DATA_BLOCK "Asse_B"	// DB 35
VERSION : 0.1
  STRUCT
   A_FD_OR : BYTE ;	//Feedrate override
   A_DriveEnable : BOOL ;	//Drive test movement enable
   A_AckFixedStop : BOOL ;	//Acknowledge fixed stop reached
   A_SensorFixedStop : BOOL ;	//Sensor fixed stop
   A_ASpDisable : BOOL ;	//Axis/spindle disable
   A_Follow_upMode : BOOL ;	//Follow-up mode
   A_PosMeas1 : BOOL ;	//Position measuring system 1
   A_PosMeas2 : BOOL ;	//Position measuring system 2
   A_ORactive : BOOL ;	//Override active
   A_SWCam : BOOL ;	//SW cam activation
   A_ContrEnable : BOOL ;	//Controller enable
   A_DelDTGSpReset : BOOL ;	//Delete distance to go/Spindle-Reset
   A_Clamp : BOOL ;	//Clamping in progress
   A_RefVal1 : BOOL ;	//Reference point value 1
   A_RefVal2 : BOOL ;	//Reference point value 2
   A_RefVal3 : BOOL ;	//Reference point value 3
   A_RefVal4 : BOOL ;	//Reference point value 4
   A_ExtZO : BOOL ;	//Import external ZO
   A_EnabTravFixedStop : BOOL ;	//Enable travel to fixed stop
   A_FixedFD1 : BOOL ;	//Activate fixed feed 1
   A_FixedFD2 : BOOL ;	//Activate fixed feed 2
   A_FixedFD3 : BOOL ;	//Activate fixed feed 3
   A_FixedFD4 : BOOL ;	//Activate fixed feed 4
   A_VelocSpeedLimit : BOOL ;	//Velocity/spindle speed limitation
   A_PrgtestAxRel : BOOL ;	// Program test axis/spindle release
   A_HW1 : BOOL ;	//Activate handwheel 1
   A_HW2 : BOOL ;	//Activate handwheel 2
   A_HW3 : BOOL ;	//Activate handwheel 3
   A_FDSpStop : BOOL ;	//Feed stop/spindle stop
   A_Disable : BOOL ;	//Traversing key disable
   A_RapidTrOR : BOOL ;	//Rapid traverse override
   A_Minus : BOOL ;	//Traversing key minus
   A_Plus : BOOL ;	//Traversing key plus
   A_INC1 : BOOL ;	//INC1
   A_INC10 : BOOL ;	//INC10
   A_INC100 : BOOL ;	//INC100
   A_INC1000 : BOOL ;	//INC1000
   A_INC10000 : BOOL ;	//INC10000
   A_INCVar : BOOL ;	//INC variable
   A_OEMAxis : BYTE ;	//OEM axis signals
   f7 : BYTE ;
   A_NCASpChanA : BOOL ;	//Assign NC axis/spindle channel A
   A_NCASpChanB : BOOL ;	//Assign NC axis/spindle channel B
   A_NCASpChanC : BOOL ;	//Assign NC axis/spindle channel C
   A_NCASpChanD : BOOL ;	//Assign NC axis/spindle channel D
   A_NCASpStrobe : BOOL ;	//Activation of assignment with pos. edge
   f8_5 : BOOL ;
   f8_6 : BOOL ;
   A_PLCASp : BOOL ;	//Request PLC axis/spindle
   A_Para_A : BOOL ;	//Parameter block servo A
   A_Para_B : BOOL ;	//Parameter block servo B
   A_Para_C : BOOL ;	//Parameter block servo C
   A_LockParSetDef : BOOL ;	//Lock parameter set definition from NC
   f9_4 : BOOL ;
   f9_5 : BOOL ;
   f9_6 : BOOL ;
   f9_7 : BOOL ;
   A_REPOSDelay : BOOL ;	//REPOS DELAY
   f10_1 : BOOL ;
   f10_2 : BOOL ;
   f10_3 : BOOL ;
   f10_4 : BOOL ;
   f10_5 : BOOL ;
   f10_6 : BOOL ;
   f10_7 : BOOL ;
   A_StartBrakeTest : BOOL ;	// Start brake test
   f11_1 : BOOL ;
   f11_2 : BOOL ;
   f11_3 : BOOL ;
   f11_4 : BOOL ;
   f11_5 : BOOL ;
   f11_6 : BOOL ;
   f11_7 : BOOL ;
   A_HWLimitMinus : BOOL ;	//Hardware limit switch minus
   A_HWLimitPlus : BOOL ;	//Hardware limit switch plus
   A_SWLimit2Minus : BOOL ;	//2nd software limit switch minus
   A_SWLimit2Plus : BOOL ;	//2nd software limit switch plus
   A_ModuloLimitEn : BOOL ;	// Modulo limit enabled
   f12_5 : BOOL ;
   f12_6 : BOOL ;
   A_DelayRef : BOOL ;	//Delay reference point approach
   f13 : BYTE ;
   f14 : INT ;
   A_ActGearA : BOOL ;	//Actual gear stage A
   A_ActGearB : BOOL ;	//Actual gear stage B
   A_ActGearC : BOOL ;	//Actual gear stage C
   A_GearChangeOv : BOOL ;	//Gear has changed over
   A_Sp1Syn : BOOL ;	//Re-synchronize spindle 1
   A_Sp2Syn : BOOL ;	//Re-synchronize spindle 2
   A_NoMonitorGear : BOOL ;	//No monitoring when changing gear
   A_DeleteS : BOOL ;	//Delete S value
   A_FD_ORSp : BOOL ;	//Feedrate override for spindle valid
   f17_1 : BOOL ;
   f17_2 : BOOL ;
   f17_3 : BOOL ;
   A_Sp1SynP : BOOL ;	//Re-synchronize spindle 1 f. positioning
   A_Sp2SynP : BOOL ;	//Re-synchronize spindle 2 f. positioning
   A_M3M4Inv : BOOL ;	//Invert M3/M4
   f17_7 : BOOL ;
   f18_0 : BOOL ;
   f18_1 : BOOL ;
   f18_2 : BOOL ;
   f18_3 : BOOL ;
   A_OscilPLC : BOOL ;	//Oscillation via PLC
   A_OscilSpeed : BOOL ;	//enable Oscillation
   A_SetRotDirectRight : BOOL ;	//Setpoint osci. direct. right
   A_SetRotDirectLeft : BOOL ;	//Setpoint osci. direct. left
   A_SpOR : BYTE ;	//Spindle override
   A_UFSwOv : BOOL ;	//Run-up switchover U/F operation
   A_RUEncQuStop : BOOL ;	//Run-up encoder quick stop
   A_Tlimit2 : BOOL ;	//Torque limit 2
   A_SpeedSetpSmooth : BOOL ;	//Speed setpoint smoothing
   f20_4 : BOOL ;
   A_HoldBrakeToOpen : BOOL ;	// holding brake open
   f20_6 : BOOL ;
   f20_7 : BOOL ;
   A_ParA : BOOL ;	//Parameter set selection A
   A_ParB : BOOL ;	//Parameter set selection B
   A_ParC : BOOL ;	//Parameter set selection C
   A_MotA : BOOL ;	//Motor selection A
   A_MotB : BOOL ;	//Motor selection B
   A_MotOK : BOOL ;	//Motor selected
   A_IntegratDisable : BOOL ;	//n controller integrator disable
   A_PulseEnable : BOOL ;	//Pulse enable
   A_SG_SBH : BOOL ;	//Deselection SG/SBH
   A_SBH : BOOL ;	//Deselection of safe standstill
   f22_2 : BOOL ;
   A_SGselect0 : BOOL ;	//Selection SG bit 0
   A_SGselect1 : BOOL ;	//Selection SG bit 1
   f22_5 : BOOL ;
   f22_6 : BOOL ;
   f22_7 : BOOL ;
   A_Transmiss0 : BOOL ;	//Selection Transmission bit 0
   A_Transmiss1 : BOOL ;	//Selection Transmission bit 1
   A_Transmiss2 : BOOL ;	//Selection Transmission bit 2
   f23_3 : BOOL ;
   A_SE : BOOL ;	//Selection SE
   A_BrakeToClose : BOOL ;	// Sinamics: Brake to close
   f23_6 : BOOL ;
   A_TestStop : BOOL ;	//Activate test stop
   A_RotationMonit : BOOL ;	// Stepper motor: Rotation monitoring
   A_ControlAx : BOOL ;	// Control Axis
   f24_2 : BOOL ;
   f24_3 : BOOL ;
   A_TorqComp : BOOL ;	// Torque compensation
   A_ChangSetpOutAss0 : BOOL ;	// Bit value for CTRLOUT_changed - Change setpoint output assignment
   A_ChangSetpOutAss1 : BOOL ;	// Bit value for CTRLOUT_changed - Change setpoint output assignment
   A_MS : BOOL ;	//Master / Slave On
   f25 : BYTE ;
   f26_0 : BOOL ;
   f26_1 : BOOL ;
   f26_2 : BOOL ;
   A_CompContr : BOOL ;	//Compensation controller On
   A_FollowAxOv : BOOL ;	//Enable following axis override
   f26_5 : BOOL ;
   f26_6 : BOOL ;
   f26_7 : BOOL ;
   A_DEPMCS : BOOL ;	// Resume: DEPMCS
   A_DEPBCS : BOOL ;	// Resume: DEPBCS
   A_Corr : BOOL ;	// Resume: Corr
   A_HIAxMove : BOOL ;	// Resume: HIAxMove
   A_StopDEPMCS : BOOL ;	// Stop: DEPMCS
   A_StopDEPBCS : BOOL ;	// Stop: DEPBCS
   A_StopCorr : BOOL ;	// Stop: Corr
   A_StopHIAxMove : BOOL ;	// Stop: HIAxMove
   A_OscillAxExtRev : BOOL ;	// OscillAxExtReversal
   A_AxReset : BOOL ;	// AXRESET
   A_AxResume : BOOL ;	// AXRESUME
   A_SetRP : BOOL ;	//Set reversal point
   A_ChangeRP : BOOL ;	//Change reversal point
   A_StopRP : BOOL ;	//Stop at next reversal point
   A_Stop : BOOL ;	//Stop
   A_PLCAxis : BOOL ;	//PLC checks axis
   f29_0 : BOOL ;
   f29_1 : BOOL ;
   f29_2 : BOOL ;
   f29_3 : BOOL ;
   A_StartGantSynRun : BOOL ;	//Start gantry synchronization run
   A_NoAutoSync : BOOL ;	//No auto sync
   f29_6 : BOOL ;
   f29_7 : BOOL ;
   A_StopSpindle : BOOL ;	//Stop spindle
   A_StartCW : BOOL ;	//Start spindle Clockwise
   A_StartCCW : BOOL ;	//Start spindle Counterclockwise
   A_AutoGearStep : BOOL ;	//Autom. gear step change
   A_PosSpindle : BOOL ;	//Position spindle
   f30_5 : BOOL ;
   f30_6 : BOOL ;
   f30_7 : BOOL ;
   f31_0 : BOOL ;
   f31_1 : BOOL ;
   f31_2 : BOOL ;
   f31_3 : BOOL ;
   A_Resynchronize : BOOL ;	// Resynchronize
   A_DisSync : BOOL ;	// Disable synchronization
   A_Tracksync : BOOL ;	// Track synchronism
   f31_7 : BOOL ;
   f32_0 : BOOL ;
   f32_1 : BOOL ;
   A_extStopA : BOOL ;	//Deselection external Stop A
   A_extStopC : BOOL ;	//Deselection external Stop C
   A_extStopD : BOOL ;	//Deselection external Stop D
   A_extStopE : BOOL ;	//Deselection external Stop E
   f32_6 : BOOL ;
   f32_7 : BOOL ;
   f33_0 : BOOL ;
   f33_1 : BOOL ;
   f33_2 : BOOL ;
   f33_3 : BOOL ;
   A_SGcorr_0 : BOOL ;	//Selection SG-correction Bit 0
   A_SGcorr_1 : BOOL ;	//Selection SG-correction Bit 1
   A_SGcorr_2 : BOOL ;	//Selection SG-correction Bit 2
   A_SGcorr_3 : BOOL ;	//Selection SG-correction Bit 3
   f34 : ARRAY  [34 .. 55 ] OF BYTE ;
   A_FeedDriveCAxEng : BOOL ;	// Seperate feed drive as C axis engaged
   A_SpSpeedDisp : BOOL ;	// Spindle speed display
   A_SpInsideClamp : BOOL ;	// Spindle inside clamping
   f56_3 : BOOL ;
   f56_4 : BOOL ;
   f56_5 : BOOL ;
   f56_6 : BOOL ;
   f56_7 : BOOL ;
   f57 : BYTE ;
   f58 : WORD ;	// FC18: internal
   E_SpNA : BOOL ;	//Spindle/no axis
   E_NCU_Link : BOOL ;	//NCU_link active axis
   E_EncodFreq1 : BOOL ;	//Encoder limit frequency 1 exceeded
   E_EncodFreq2 : BOOL ;	//Encoder limit frequency 2 exceeded
   E_RefSyn1 : BOOL ;	//Referenced/synchronized 1
   E_RefSyn2 : BOOL ;	//Referenced/synchronized 2
   E_ExactCoarse : BOOL ;	//Position reached with exact stop coarse
   E_ExactFine : BOOL ;	//Position reached with exact stop fine
   E_TravRequ : BOOL ;	//Travel request
   E_AxialAlarm : BOOL ;	// Axial alarm
   E_AxisReady : BOOL ;	//Axis ready
   E_Follow_upMode : BOOL ;	//Follow-up mode active
   E_Stat : BOOL ;	//Axis/spindle stationary (n<nmin)
   E_PositContr : BOOL ;	//Position controller active
   E_SpeedContr : BOOL ;	//Speed controller active
   E_CurrentContr : BOOL ;	//Current controller active
   E_SWCam : BOOL ;	//Software cams active
   E_HWOverlay : BOOL ;	//Handwheel overlay active
   E_RevFD : BOOL ;	//Revolutional feedrate active
   E_MeasAct : BOOL ;	//Measuring active
   E_ActTravFStop : BOOL ;	//Activate travel to fixed stop
   E_FixedStop : BOOL ;	//Fixed stop reached
   E_ForceFixedStop : BOOL ;	// Force fixed stop limited
   E_AxContainerRot : BOOL ;	// Axis container rotation active
   E_AxReset : BOOL ;	// Axis reset done
   E_PLCCtrlAx : BOOL ;	// PLCcontrolled axis
   E_AxStop : BOOL ;	// Axis stop active
   E_AxSpDisable : BOOL ;	// Axis/spindle disable active
   E_StopDEPMCS : BOOL ;	// stop DEPMCS active
   E_StopDEPBCS : BOOL ;	// stop DEPBCS active
   E_StopCorr : BOOL ;	// stop Corr active
   E_StopHIAxMove : BOOL ;	// Stop HIAxMove active
   E_HW1 : BOOL ;	//Handwheel 1 active
   E_HW2 : BOOL ;	//Handwheel 2 active
   E_HW3 : BOOL ;	//Handwheel 3 active
   f64_3 : BOOL ;
   E_TReqMinus : BOOL ;	// Travel request minus
   E_TReqPlus : BOOL ;	// Travel request plus
   E_TCMinus : BOOL ;	//Traverse command minus
   E_TCPlus : BOOL ;	//Traverse command plus
   E_INC1 : BOOL ;	//INC1
   E_INC10 : BOOL ;	//INC10
   E_INC100 : BOOL ;	//INC100
   E_INC1000 : BOOL ;	//INC1000
   E_INC10000 : BOOL ;	//INC10000
   E_INCVar : BOOL ;	//INC variable
   f65_6 : BOOL ;
   f65_7 : BOOL ;
   E_OEMAxis : BYTE ;	//OEM axis signals
   f67 : BYTE ;
   E_NCASpChanA : BOOL ;	//NC axis/spindle in channel A
   E_NCASpChanB : BOOL ;	//NC axis/spindle in channel B
   E_NCASpChanC : BOOL ;	//NC axis/spindle in channel C
   E_NCASpChanD : BOOL ;	//NC axis/spindle in channel D
   E_PLCType : BOOL ;	//New type requested by PLC
   E_ChPoss : BOOL ;	//Change axis possible
   E_NeutrASp : BOOL ;	//Neutral axis/spindle
   E_PLCASp : BOOL ;	//PLC axis/spindle
   E_ParS_A : BOOL ;	//Parameter block servo A
   E_ParS_B : BOOL ;	//Parameter block servo B
   E_ParS_C : BOOL ;	//Parameter block servo C
   E_ReposSh : BOOL ;	// Repos shift
   E_ReposShValid : BOOL ;	// Repos shift valid
   E_ReposDelayQuit : BOOL ;	// Repos delay quit
   f70_3 : BOOL ;
   f70_4 : BOOL ;
   f70_5 : BOOL ;
   f70_6 : BOOL ;
   f70_7 : BOOL ;
   E_BrakeTest : BOOL ;	// Brake test active
   f71_1 : BOOL ;
   f71_2 : BOOL ;
   f71_3 : BOOL ;
   f71_4 : BOOL ;
   f71_5 : BOOL ;
   f71_6 : BOOL ;
   E_PLCAxDedic : BOOL ;	// PLC Axis dedicated
   E_MMC_REPOSDelay : BOOL ;	//MMC REPOS DELAY
   f72_1 : BOOL ;
   f72_2 : BOOL ;
   f72_3 : BOOL ;
   f72_4 : BOOL ;
   f72_5 : BOOL ;
   f72_6 : BOOL ;
   f72_7 : BOOL ;
   f73 : BYTE ;
   f74_0 : BOOL ;
   f74_1 : BOOL ;
   f74_2 : BOOL ;
   f74_3 : BOOL ;
   E_ModLimEnAct : BOOL ;	// Modulo limit enabled active
   f74_5 : BOOL ;
   f74_6 : BOOL ;
   f74_7 : BOOL ;
   f75 : BYTE ;
   E_ScratchPulse : BOOL ;	//Scratch pulse
   f76_1 : BOOL ;
   f76_2 : BOOL ;
   f76_3 : BOOL ;
   E_PathAxis : BOOL ;	// Path axis
   E_PosAxis : BOOL ;	//Positioning axis
   E_IndexAxisPos : BOOL ;	//Indexing axis in position
   E_CurvePos : BOOL ;	//Curve axis in position
   E_CollCheckRedSpeed : BOOL ;	//reduced speed of Collisions Check
   f77_1 : BOOL ;
   f77_2 : BOOL ;
   f77_3 : BOOL ;
   f77_4 : BOOL ;
   f77_5 : BOOL ;
   f77_6 : BOOL ;
   f77_7 : BOOL ;
   E_FPosAxis : REAL ;	//F function (REAL format) for positioning axes
   E_SetpGearA : BOOL ;	//Setpoint gear stage A
   E_SetpGearB : BOOL ;	//Setpoint gear stage B
   E_SetpGearC : BOOL ;	//Setpoint gear stage C
   E_GearChange : BOOL ;	//Gear changeover
   f82_4 : BOOL ;
   f82_5 : BOOL ;
   f82_6 : BOOL ;
   f82_7 : BOOL ;
   E_SpeedLimit : BOOL ;	//Speed limit exceeded
   E_SetSpeedLimit : BOOL ;	//Setpoint speed limited
   E_SetSpeedIncreased : BOOL ;	//Setpoint speed increased
   E_GeoMonit : BOOL ;	//Geometry monitoring
   E_SupportAreaViol : BOOL ;	//Support area limits violated
   E_SetRange : BOOL ;	//Spindle in setpoint range
   E_SpeedMonit : BOOL ;	//Speed monitoring
   E_ActRotRight : BOOL ;	//Actual rotation direction right
   E_ConstCuttSpeed : BOOL ;	//Const. cutting speed active
   E_SUG : BOOL ;	//SUG active (grinding wheel surface speed)
   E_CLG : BOOL ;	//CLG active
   E_Tapping : BOOL ;	//Tapping without compensating chuck
   E_SyncMode : BOOL ;	//Synchronous mode spindle active
   E_PosMode : BOOL ;	//Positioning mode spindle active
   E_OscillMode : BOOL ;	//Oscillation mode spindle active
   E_ContrMode : BOOL ;	//Control mode spindle active
   f85_0 : BOOL ;
   f85_1 : BOOL ;
   f85_2 : BOOL ;
   f85_3 : BOOL ;
   f85_4 : BOOL ;
   E_SpInPosition : BOOL ;	// Spindle in position
   f85_6 : BOOL ;
   f85_7 : BOOL ;
   E_MFunct : INT ;	//M function (INT) for spindle
   E_SFunct : REAL ;	//S function (REAL) for spindle
   E_SetUpMode : BOOL ;	//Set-up mode active
   E_RUEncDisabl : BOOL ;	//Run-up encoder disable active
   E_Tlimit2 : BOOL ;	//Torque limit 2 active
   E_SpeedSetpSmooth : BOOL ;	//Speed setpoint smoothing active
   E_RLIact : BOOL ;	// RLI active
   E_HoldBrakeOpened : BOOL ;	// holding brake opened
   E_EarthFaultDetec : BOOL ;	// earth-fault detection
   f92_7 : BOOL ;
   E_ParA : BOOL ;	//Active parameter set A
   E_ParB : BOOL ;	//Active parameter set B
   E_ParC : BOOL ;	//Active parameter set C
   E_MotA : BOOL ;	//Active motor A
   E_MotB : BOOL ;	//Active motor B
   E_MotOK : BOOL ;	//Drive ready
   E_IntegratDisable : BOOL ;	//n controller integrator disabled
   E_PulseEnable : BOOL ;	//Pulses enabled
   E_MTempWarn : BOOL ;	//Temperature prewarning motor
   E_HTempWarn : BOOL ;	//Temperature prewarning heat sink
   E_RUComplete : BOOL ;	//Ramp-up complete
   E_MdMdx : BOOL ;	//Md<Mdx
   E_NactNmin : BOOL ;	//nact<nmin
   E_NactNx : BOOL ;	//nact<nx
   E_NactNset : BOOL ;	//nact<nset
   E_Message : BOOL ;	//Variable message function
   E_UDClessAlThreshold : BOOL ;	//UDC-link < alarm threshold
   E_RetractVolt : BOOL ;	// Fall short of retract voltage
   E_Generator : BOOL ;	// Generator active
   E_MinGeneratorVolt : BOOL ;	// Fall short of min. generator voltage
   E_SpeedThreshold : BOOL ;	// Speed threshold star/delta
   f95_5 : BOOL ;
   f95_6 : BOOL ;
   E_PowerSecI2TLimit : BOOL ;	// Power Section I2T limit
   E_SpindleMonit : BOOL ;	//Error spindle monitoring
   E_AxisCtrl : BOOL ;	// Axis control active
   E_MSFine : BOOL ;	// Master/Slave fine
   E_MSCoarse : BOOL ;	// Master/Slave coarse
   E_MSCompContr : BOOL ;	// Master/Slave Compensation controller activ
   E_BitValCtrlOutChang0 : BOOL ;	// Bit value for CTRLOUT_changed 0:  Change setpoint output assignment
   E_BitValCtrlOutChang1 : BOOL ;	// Bit value for CTRLOUT_changed 1:  Change setpoint output assignment
   E_MS : BOOL ;	//Master/ slave active
   f97 : BYTE ;
   E_SyncronFine : BOOL ;	//Synchronism fine
   E_SyncronCoarse : BOOL ;	//Synchronism coarse
   E_ActValCoupling : BOOL ;	//Actual value coupling
   f98_3 : BOOL ;
   E_OverlayMotion : BOOL ;	//Overlaid motion
   E_SWL : BOOL ;	//Speed warning limit reached
   E_AWL : BOOL ;	//Acceleration warning limit reached
   E_EmRetr : BOOL ;	//Emergency retraction active
   E_MasterSp : BOOL ;	//Master spindle
   E_SlaveSp : BOOL ;	//Slave spindle
   f99_2 : BOOL ;
   E_AxisAccel : BOOL ;	//Axis accelerated
   E_Sync : BOOL ;	//Synchronization active
   E_MSR : BOOL ;	//Max speed reached
   E_MAR : BOOL ;	//Max acceleration reached
   E_EmRetrEnabl : BOOL ;	//Emergency retraction enabled
   f100_0 : BOOL ;
   f100_1 : BOOL ;
   E_OscillAxExtRev : BOOL ;	// OscillAxExt Reversal active
   E_StopOscill : BOOL ;	//Oscillation cannot start
   E_ErrorOscill : BOOL ;	//Error during oscillation
   E_SparkOut : BOOL ;	//Spark-out active
   E_OscillMotion : BOOL ;	//Oscillation motion active
   E_Oscill : BOOL ;	//Oscillation active
   f101_0 : BOOL ;
   f101_1 : BOOL ;
   E_GantCOLimit : BOOL ;	//Gantry cut-off limit exceeded
   E_GantWarn : BOOL ;	//Gantry warning limit exceeded
   E_SynRunStart : BOOL ;	//Synchronization run ready to start
   E_GantGroupSyn : BOOL ;	//Gantry grouping is synchronous
   E_GantLeadAxis : BOOL ;	//Gantry leading axis
   E_GantAxis : BOOL ;	//Gantry axis
   f102 : INT ;
   E_AIAxis : ARRAY  [1 .. 31 ] OF BOOL ;	//Active infeed axis[1..31]
   E_SG_SBH : BOOL ;	//Active SG/SBH
   E_ErrLifeS_CRC : BOOL ;	// Error lifesign or CRC-error
   E_ImpdelNCK : BOOL ;	//Delete pulses NCK
   r108_3 : BOOL ;
   r108_4 : BOOL ;
   r108_5 : BOOL ;
   E_SE2 : BOOL ;	//SE 2 active
   E_SRef : BOOL ;	//Axis safely referenced
   E_SN1Plus : BOOL ;	//Actual position > cam position SN1+
   E_SN1Minus : BOOL ;	//Actual position > cam position SN1-
   E_SN2Plus : BOOL ;	//Actual position > cam position SN2+
   E_SN2Minus : BOOL ;	//Actual position > cam position SN2-
   E_SN3Plus : BOOL ;	//Actual position > cam position SN3+
   E_SN3Minus : BOOL ;	//Actual position > cam position SN3-
   E_SN4Plus : BOOL ;	//Actual position > cam position SN4+
   E_SN4Minus : BOOL ;	//Actual position > cam position SN4-
   f110_0 : BOOL ;
   E_SBH : BOOL ;	//Active SBH
   f110_2 : BOOL ;
   E_SG_0 : BOOL ;	//Active SG 0
   E_SG_1 : BOOL ;	//Active SG 1
   E_n_nx : BOOL ;	//n < nx
   f110_6 : BOOL ;
   f110_7 : BOOL ;
   f111_0 : BOOL ;
   f111_1 : BOOL ;
   f111_2 : BOOL ;
   f111_3 : BOOL ;
   E_StopAB : BOOL ;	//Stop A/B active
   E_StopC : BOOL ;	//Stop C active
   E_StopD : BOOL ;	//Stop D active
   E_StopE : BOOL ;	//Stop E active
   E_CamRangeTr1 : BYTE ;	//Cam Range for Cam Track 1
   E_CamRangeTr2 : BYTE ;	//Cam Range for Cam Track 2
   E_CamRangeTr3 : BYTE ;	//Cam Range for Cam Track 3
   E_CamRangeTr4 : BYTE ;	//Cam Range for Cam Track 4
   f116 : BYTE ;
   E_CamTrack1 : BOOL ;	//Cam Track 1
   E_CamTrack2 : BOOL ;	//Cam Track 2
   E_CamTrack3 : BOOL ;	//Cam Track 3
   E_CamTrack4 : BOOL ;	//Cam Track 4
   f117_4 : BOOL ;
   f117_5 : BOOL ;
   f117_6 : BOOL ;
   f117_7 : BOOL ;
   E_CamRangeBitTr1 : ARRAY  [0 .. 14 ] OF //Cam Range Bits for Cam Track 1
   BOOL ;
   E_CamRangeBitTr2 : ARRAY  [0 .. 14 ] OF //Cam Range Bits for Cam Track 2
   BOOL ;
   E_CamRangeBitTr3 : ARRAY  [0 .. 14 ] OF //Cam Range Bits for Cam Track 3
   BOOL ;
   E_CamRangeBitTr4 : ARRAY  [0 .. 14 ] OF //Cam Range Bits for Cam Track 4
   BOOL ;
  END_STRUCT ;	
BEGIN
END_DATA_BLOCK

DATA_BLOCK "Asse_Mandrino"	// DB 36
VERSION : 0.1
  STRUCT
   A_FD_OR : BYTE ;	//Feedrate override
   A_DriveEnable : BOOL ;	//Drive test movement enable
   A_AckFixedStop : BOOL ;	//Acknowledge fixed stop reached
   A_SensorFixedStop : BOOL ;	//Sensor fixed stop
   A_ASpDisable : BOOL ;	//Axis/spindle disable
   A_Follow_upMode : BOOL ;	//Follow-up mode
   A_PosMeas1 : BOOL ;	//Position measuring system 1
   A_PosMeas2 : BOOL ;	//Position measuring system 2
   A_ORactive : BOOL ;	//Override active
   A_SWCam : BOOL ;	//SW cam activation
   A_ContrEnable : BOOL ;	//Controller enable
   A_DelDTGSpReset : BOOL ;	//Delete distance to go/Spindle-Reset
   A_Clamp : BOOL ;	//Clamping in progress
   A_RefVal1 : BOOL ;	//Reference point value 1
   A_RefVal2 : BOOL ;	//Reference point value 2
   A_RefVal3 : BOOL ;	//Reference point value 3
   A_RefVal4 : BOOL ;	//Reference point value 4
   A_ExtZO : BOOL ;	//Import external ZO
   A_EnabTravFixedStop : BOOL ;	//Enable travel to fixed stop
   A_FixedFD1 : BOOL ;	//Activate fixed feed 1
   A_FixedFD2 : BOOL ;	//Activate fixed feed 2
   A_FixedFD3 : BOOL ;	//Activate fixed feed 3
   A_FixedFD4 : BOOL ;	//Activate fixed feed 4
   A_VelocSpeedLimit : BOOL ;	//Velocity/spindle speed limitation
   A_PrgtestAxRel : BOOL ;	// Program test axis/spindle release
   A_HW1 : BOOL ;	//Activate handwheel 1
   A_HW2 : BOOL ;	//Activate handwheel 2
   A_HW3 : BOOL ;	//Activate handwheel 3
   A_FDSpStop : BOOL ;	//Feed stop/spindle stop
   A_Disable : BOOL ;	//Traversing key disable
   A_RapidTrOR : BOOL ;	//Rapid traverse override
   A_Minus : BOOL ;	//Traversing key minus
   A_Plus : BOOL ;	//Traversing key plus
   A_INC1 : BOOL ;	//INC1
   A_INC10 : BOOL ;	//INC10
   A_INC100 : BOOL ;	//INC100
   A_INC1000 : BOOL ;	//INC1000
   A_INC10000 : BOOL ;	//INC10000
   A_INCVar : BOOL ;	//INC variable
   A_OEMAxis : BYTE ;	//OEM axis signals
   f7 : BYTE ;
   A_NCASpChanA : BOOL ;	//Assign NC axis/spindle channel A
   A_NCASpChanB : BOOL ;	//Assign NC axis/spindle channel B
   A_NCASpChanC : BOOL ;	//Assign NC axis/spindle channel C
   A_NCASpChanD : BOOL ;	//Assign NC axis/spindle channel D
   A_NCASpStrobe : BOOL ;	//Activation of assignment with pos. edge
   f8_5 : BOOL ;
   f8_6 : BOOL ;
   A_PLCASp : BOOL ;	//Request PLC axis/spindle
   A_Para_A : BOOL ;	//Parameter block servo A
   A_Para_B : BOOL ;	//Parameter block servo B
   A_Para_C : BOOL ;	//Parameter block servo C
   A_LockParSetDef : BOOL ;	//Lock parameter set definition from NC
   f9_4 : BOOL ;
   f9_5 : BOOL ;
   f9_6 : BOOL ;
   f9_7 : BOOL ;
   A_REPOSDelay : BOOL ;	//REPOS DELAY
   f10_1 : BOOL ;
   f10_2 : BOOL ;
   f10_3 : BOOL ;
   f10_4 : BOOL ;
   f10_5 : BOOL ;
   f10_6 : BOOL ;
   f10_7 : BOOL ;
   A_StartBrakeTest : BOOL ;	// Start brake test
   f11_1 : BOOL ;
   f11_2 : BOOL ;
   f11_3 : BOOL ;
   f11_4 : BOOL ;
   f11_5 : BOOL ;
   f11_6 : BOOL ;
   f11_7 : BOOL ;
   A_HWLimitMinus : BOOL ;	//Hardware limit switch minus
   A_HWLimitPlus : BOOL ;	//Hardware limit switch plus
   A_SWLimit2Minus : BOOL ;	//2nd software limit switch minus
   A_SWLimit2Plus : BOOL ;	//2nd software limit switch plus
   A_ModuloLimitEn : BOOL ;	// Modulo limit enabled
   f12_5 : BOOL ;
   f12_6 : BOOL ;
   A_DelayRef : BOOL ;	//Delay reference point approach
   f13 : BYTE ;
   f14 : INT ;
   A_ActGearA : BOOL ;	//Actual gear stage A
   A_ActGearB : BOOL ;	//Actual gear stage B
   A_ActGearC : BOOL ;	//Actual gear stage C
   A_GearChangeOv : BOOL ;	//Gear has changed over
   A_Sp1Syn : BOOL ;	//Re-synchronize spindle 1
   A_Sp2Syn : BOOL ;	//Re-synchronize spindle 2
   A_NoMonitorGear : BOOL ;	//No monitoring when changing gear
   A_DeleteS : BOOL ;	//Delete S value
   A_FD_ORSp : BOOL ;	//Feedrate override for spindle valid
   f17_1 : BOOL ;
   f17_2 : BOOL ;
   f17_3 : BOOL ;
   A_Sp1SynP : BOOL ;	//Re-synchronize spindle 1 f. positioning
   A_Sp2SynP : BOOL ;	//Re-synchronize spindle 2 f. positioning
   A_M3M4Inv : BOOL ;	//Invert M3/M4
   f17_7 : BOOL ;
   f18_0 : BOOL ;
   f18_1 : BOOL ;
   f18_2 : BOOL ;
   f18_3 : BOOL ;
   A_OscilPLC : BOOL ;	//Oscillation via PLC
   A_OscilSpeed : BOOL ;	//enable Oscillation
   A_SetRotDirectRight : BOOL ;	//Setpoint osci. direct. right
   A_SetRotDirectLeft : BOOL ;	//Setpoint osci. direct. left
   A_SpOR : BYTE ;	//Spindle override
   A_UFSwOv : BOOL ;	//Run-up switchover U/F operation
   A_RUEncQuStop : BOOL ;	//Run-up encoder quick stop
   A_Tlimit2 : BOOL ;	//Torque limit 2
   A_SpeedSetpSmooth : BOOL ;	//Speed setpoint smoothing
   f20_4 : BOOL ;
   A_HoldBrakeToOpen : BOOL ;	// holding brake open
   f20_6 : BOOL ;
   f20_7 : BOOL ;
   A_ParA : BOOL ;	//Parameter set selection A
   A_ParB : BOOL ;	//Parameter set selection B
   A_ParC : BOOL ;	//Parameter set selection C
   A_MotA : BOOL ;	//Motor selection A
   A_MotB : BOOL ;	//Motor selection B
   A_MotOK : BOOL ;	//Motor selected
   A_IntegratDisable : BOOL ;	//n controller integrator disable
   A_PulseEnable : BOOL ;	//Pulse enable
   A_SG_SBH : BOOL ;	//Deselection SG/SBH
   A_SBH : BOOL ;	//Deselection of safe standstill
   f22_2 : BOOL ;
   A_SGselect0 : BOOL ;	//Selection SG bit 0
   A_SGselect1 : BOOL ;	//Selection SG bit 1
   f22_5 : BOOL ;
   f22_6 : BOOL ;
   f22_7 : BOOL ;
   A_Transmiss0 : BOOL ;	//Selection Transmission bit 0
   A_Transmiss1 : BOOL ;	//Selection Transmission bit 1
   A_Transmiss2 : BOOL ;	//Selection Transmission bit 2
   f23_3 : BOOL ;
   A_SE : BOOL ;	//Selection SE
   A_BrakeToClose : BOOL ;	// Sinamics: Brake to close
   f23_6 : BOOL ;
   A_TestStop : BOOL ;	//Activate test stop
   A_RotationMonit : BOOL ;	// Stepper motor: Rotation monitoring
   A_ControlAx : BOOL ;	// Control Axis
   f24_2 : BOOL ;
   f24_3 : BOOL ;
   A_TorqComp : BOOL ;	// Torque compensation
   A_ChangSetpOutAss0 : BOOL ;	// Bit value for CTRLOUT_changed - Change setpoint output assignment
   A_ChangSetpOutAss1 : BOOL ;	// Bit value for CTRLOUT_changed - Change setpoint output assignment
   A_MS : BOOL ;	//Master / Slave On
   f25 : BYTE ;
   f26_0 : BOOL ;
   f26_1 : BOOL ;
   f26_2 : BOOL ;
   A_CompContr : BOOL ;	//Compensation controller On
   A_FollowAxOv : BOOL ;	//Enable following axis override
   f26_5 : BOOL ;
   f26_6 : BOOL ;
   f26_7 : BOOL ;
   A_DEPMCS : BOOL ;	// Resume: DEPMCS
   A_DEPBCS : BOOL ;	// Resume: DEPBCS
   A_Corr : BOOL ;	// Resume: Corr
   A_HIAxMove : BOOL ;	// Resume: HIAxMove
   A_StopDEPMCS : BOOL ;	// Stop: DEPMCS
   A_StopDEPBCS : BOOL ;	// Stop: DEPBCS
   A_StopCorr : BOOL ;	// Stop: Corr
   A_StopHIAxMove : BOOL ;	// Stop: HIAxMove
   A_OscillAxExtRev : BOOL ;	// OscillAxExtReversal
   A_AxReset : BOOL ;	// AXRESET
   A_AxResume : BOOL ;	// AXRESUME
   A_SetRP : BOOL ;	//Set reversal point
   A_ChangeRP : BOOL ;	//Change reversal point
   A_StopRP : BOOL ;	//Stop at next reversal point
   A_Stop : BOOL ;	//Stop
   A_PLCAxis : BOOL ;	//PLC checks axis
   f29_0 : BOOL ;
   f29_1 : BOOL ;
   f29_2 : BOOL ;
   f29_3 : BOOL ;
   A_StartGantSynRun : BOOL ;	//Start gantry synchronization run
   A_NoAutoSync : BOOL ;	//No auto sync
   f29_6 : BOOL ;
   f29_7 : BOOL ;
   A_StopSpindle : BOOL ;	//Stop spindle
   A_StartCW : BOOL ;	//Start spindle Clockwise
   A_StartCCW : BOOL ;	//Start spindle Counterclockwise
   A_AutoGearStep : BOOL ;	//Autom. gear step change
   A_PosSpindle : BOOL ;	//Position spindle
   f30_5 : BOOL ;
   f30_6 : BOOL ;
   f30_7 : BOOL ;
   f31_0 : BOOL ;
   f31_1 : BOOL ;
   f31_2 : BOOL ;
   f31_3 : BOOL ;
   A_Resynchronize : BOOL ;	// Resynchronize
   A_DisSync : BOOL ;	// Disable synchronization
   A_Tracksync : BOOL ;	// Track synchronism
   f31_7 : BOOL ;
   f32_0 : BOOL ;
   f32_1 : BOOL ;
   A_extStopA : BOOL ;	//Deselection external Stop A
   A_extStopC : BOOL ;	//Deselection external Stop C
   A_extStopD : BOOL ;	//Deselection external Stop D
   A_extStopE : BOOL ;	//Deselection external Stop E
   f32_6 : BOOL ;
   f32_7 : BOOL ;
   f33_0 : BOOL ;
   f33_1 : BOOL ;
   f33_2 : BOOL ;
   f33_3 : BOOL ;
   A_SGcorr_0 : BOOL ;	//Selection SG-correction Bit 0
   A_SGcorr_1 : BOOL ;	//Selection SG-correction Bit 1
   A_SGcorr_2 : BOOL ;	//Selection SG-correction Bit 2
   A_SGcorr_3 : BOOL ;	//Selection SG-correction Bit 3
   f34 : ARRAY  [34 .. 55 ] OF BYTE ;
   A_FeedDriveCAxEng : BOOL ;	// Seperate feed drive as C axis engaged
   A_SpSpeedDisp : BOOL ;	// Spindle speed display
   A_SpInsideClamp : BOOL ;	// Spindle inside clamping
   f56_3 : BOOL ;
   f56_4 : BOOL ;
   f56_5 : BOOL ;
   f56_6 : BOOL ;
   f56_7 : BOOL ;
   f57 : BYTE ;
   f58 : WORD ;	// FC18: internal
   E_SpNA : BOOL ;	//Spindle/no axis
   E_NCU_Link : BOOL ;	//NCU_link active axis
   E_EncodFreq1 : BOOL ;	//Encoder limit frequency 1 exceeded
   E_EncodFreq2 : BOOL ;	//Encoder limit frequency 2 exceeded
   E_RefSyn1 : BOOL ;	//Referenced/synchronized 1
   E_RefSyn2 : BOOL ;	//Referenced/synchronized 2
   E_ExactCoarse : BOOL ;	//Position reached with exact stop coarse
   E_ExactFine : BOOL ;	//Position reached with exact stop fine
   E_TravRequ : BOOL ;	//Travel request
   E_AxialAlarm : BOOL ;	// Axial alarm
   E_AxisReady : BOOL ;	//Axis ready
   E_Follow_upMode : BOOL ;	//Follow-up mode active
   E_Stat : BOOL ;	//Axis/spindle stationary (n<nmin)
   E_PositContr : BOOL ;	//Position controller active
   E_SpeedContr : BOOL ;	//Speed controller active
   E_CurrentContr : BOOL ;	//Current controller active
   E_SWCam : BOOL ;	//Software cams active
   E_HWOverlay : BOOL ;	//Handwheel overlay active
   E_RevFD : BOOL ;	//Revolutional feedrate active
   E_MeasAct : BOOL ;	//Measuring active
   E_ActTravFStop : BOOL ;	//Activate travel to fixed stop
   E_FixedStop : BOOL ;	//Fixed stop reached
   E_ForceFixedStop : BOOL ;	// Force fixed stop limited
   E_AxContainerRot : BOOL ;	// Axis container rotation active
   E_AxReset : BOOL ;	// Axis reset done
   E_PLCCtrlAx : BOOL ;	// PLCcontrolled axis
   E_AxStop : BOOL ;	// Axis stop active
   E_AxSpDisable : BOOL ;	// Axis/spindle disable active
   E_StopDEPMCS : BOOL ;	// stop DEPMCS active
   E_StopDEPBCS : BOOL ;	// stop DEPBCS active
   E_StopCorr : BOOL ;	// stop Corr active
   E_StopHIAxMove : BOOL ;	// Stop HIAxMove active
   E_HW1 : BOOL ;	//Handwheel 1 active
   E_HW2 : BOOL ;	//Handwheel 2 active
   E_HW3 : BOOL ;	//Handwheel 3 active
   f64_3 : BOOL ;
   E_TReqMinus : BOOL ;	// Travel request minus
   E_TReqPlus : BOOL ;	// Travel request plus
   E_TCMinus : BOOL ;	//Traverse command minus
   E_TCPlus : BOOL ;	//Traverse command plus
   E_INC1 : BOOL ;	//INC1
   E_INC10 : BOOL ;	//INC10
   E_INC100 : BOOL ;	//INC100
   E_INC1000 : BOOL ;	//INC1000
   E_INC10000 : BOOL ;	//INC10000
   E_INCVar : BOOL ;	//INC variable
   f65_6 : BOOL ;
   f65_7 : BOOL ;
   E_OEMAxis : BYTE ;	//OEM axis signals
   f67 : BYTE ;
   E_NCASpChanA : BOOL ;	//NC axis/spindle in channel A
   E_NCASpChanB : BOOL ;	//NC axis/spindle in channel B
   E_NCASpChanC : BOOL ;	//NC axis/spindle in channel C
   E_NCASpChanD : BOOL ;	//NC axis/spindle in channel D
   E_PLCType : BOOL ;	//New type requested by PLC
   E_ChPoss : BOOL ;	//Change axis possible
   E_NeutrASp : BOOL ;	//Neutral axis/spindle
   E_PLCASp : BOOL ;	//PLC axis/spindle
   E_ParS_A : BOOL ;	//Parameter block servo A
   E_ParS_B : BOOL ;	//Parameter block servo B
   E_ParS_C : BOOL ;	//Parameter block servo C
   E_ReposSh : BOOL ;	// Repos shift
   E_ReposShValid : BOOL ;	// Repos shift valid
   E_ReposDelayQuit : BOOL ;	// Repos delay quit
   f70_3 : BOOL ;
   f70_4 : BOOL ;
   f70_5 : BOOL ;
   f70_6 : BOOL ;
   f70_7 : BOOL ;
   E_BrakeTest : BOOL ;	// Brake test active
   f71_1 : BOOL ;
   f71_2 : BOOL ;
   f71_3 : BOOL ;
   f71_4 : BOOL ;
   f71_5 : BOOL ;
   f71_6 : BOOL ;
   E_PLCAxDedic : BOOL ;	// PLC Axis dedicated
   E_MMC_REPOSDelay : BOOL ;	//MMC REPOS DELAY
   f72_1 : BOOL ;
   f72_2 : BOOL ;
   f72_3 : BOOL ;
   f72_4 : BOOL ;
   f72_5 : BOOL ;
   f72_6 : BOOL ;
   f72_7 : BOOL ;
   f73 : BYTE ;
   f74_0 : BOOL ;
   f74_1 : BOOL ;
   f74_2 : BOOL ;
   f74_3 : BOOL ;
   E_ModLimEnAct : BOOL ;	// Modulo limit enabled active
   f74_5 : BOOL ;
   f74_6 : BOOL ;
   f74_7 : BOOL ;
   f75 : BYTE ;
   E_ScratchPulse : BOOL ;	//Scratch pulse
   f76_1 : BOOL ;
   f76_2 : BOOL ;
   f76_3 : BOOL ;
   E_PathAxis : BOOL ;	// Path axis
   E_PosAxis : BOOL ;	//Positioning axis
   E_IndexAxisPos : BOOL ;	//Indexing axis in position
   E_CurvePos : BOOL ;	//Curve axis in position
   E_CollCheckRedSpeed : BOOL ;	//reduced speed of Collisions Check
   f77_1 : BOOL ;
   f77_2 : BOOL ;
   f77_3 : BOOL ;
   f77_4 : BOOL ;
   f77_5 : BOOL ;
   f77_6 : BOOL ;
   f77_7 : BOOL ;
   E_FPosAxis : REAL ;	//F function (REAL format) for positioning axes
   E_SetpGearA : BOOL ;	//Setpoint gear stage A
   E_SetpGearB : BOOL ;	//Setpoint gear stage B
   E_SetpGearC : BOOL ;	//Setpoint gear stage C
   E_GearChange : BOOL ;	//Gear changeover
   f82_4 : BOOL ;
   f82_5 : BOOL ;
   f82_6 : BOOL ;
   f82_7 : BOOL ;
   E_SpeedLimit : BOOL ;	//Speed limit exceeded
   E_SetSpeedLimit : BOOL ;	//Setpoint speed limited
   E_SetSpeedIncreased : BOOL ;	//Setpoint speed increased
   E_GeoMonit : BOOL ;	//Geometry monitoring
   E_SupportAreaViol : BOOL ;	//Support area limits violated
   E_SetRange : BOOL ;	//Spindle in setpoint range
   E_SpeedMonit : BOOL ;	//Speed monitoring
   E_ActRotRight : BOOL ;	//Actual rotation direction right
   E_ConstCuttSpeed : BOOL ;	//Const. cutting speed active
   E_SUG : BOOL ;	//SUG active (grinding wheel surface speed)
   E_CLG : BOOL ;	//CLG active
   E_Tapping : BOOL ;	//Tapping without compensating chuck
   E_SyncMode : BOOL ;	//Synchronous mode spindle active
   E_PosMode : BOOL ;	//Positioning mode spindle active
   E_OscillMode : BOOL ;	//Oscillation mode spindle active
   E_ContrMode : BOOL ;	//Control mode spindle active
   f85_0 : BOOL ;
   f85_1 : BOOL ;
   f85_2 : BOOL ;
   f85_3 : BOOL ;
   f85_4 : BOOL ;
   E_SpInPosition : BOOL ;	// Spindle in position
   f85_6 : BOOL ;
   f85_7 : BOOL ;
   E_MFunct : INT ;	//M function (INT) for spindle
   E_SFunct : REAL ;	//S function (REAL) for spindle
   E_SetUpMode : BOOL ;	//Set-up mode active
   E_RUEncDisabl : BOOL ;	//Run-up encoder disable active
   E_Tlimit2 : BOOL ;	//Torque limit 2 active
   E_SpeedSetpSmooth : BOOL ;	//Speed setpoint smoothing active
   E_RLIact : BOOL ;	// RLI active
   E_HoldBrakeOpened : BOOL ;	// holding brake opened
   E_EarthFaultDetec : BOOL ;	// earth-fault detection
   f92_7 : BOOL ;
   E_ParA : BOOL ;	//Active parameter set A
   E_ParB : BOOL ;	//Active parameter set B
   E_ParC : BOOL ;	//Active parameter set C
   E_MotA : BOOL ;	//Active motor A
   E_MotB : BOOL ;	//Active motor B
   E_MotOK : BOOL ;	//Drive ready
   E_IntegratDisable : BOOL ;	//n controller integrator disabled
   E_PulseEnable : BOOL ;	//Pulses enabled
   E_MTempWarn : BOOL ;	//Temperature prewarning motor
   E_HTempWarn : BOOL ;	//Temperature prewarning heat sink
   E_RUComplete : BOOL ;	//Ramp-up complete
   E_MdMdx : BOOL ;	//Md<Mdx
   E_NactNmin : BOOL ;	//nact<nmin
   E_NactNx : BOOL ;	//nact<nx
   E_NactNset : BOOL ;	//nact<nset
   E_Message : BOOL ;	//Variable message function
   E_UDClessAlThreshold : BOOL ;	//UDC-link < alarm threshold
   E_RetractVolt : BOOL ;	// Fall short of retract voltage
   E_Generator : BOOL ;	// Generator active
   E_MinGeneratorVolt : BOOL ;	// Fall short of min. generator voltage
   E_SpeedThreshold : BOOL ;	// Speed threshold star/delta
   f95_5 : BOOL ;
   f95_6 : BOOL ;
   E_PowerSecI2TLimit : BOOL ;	// Power Section I2T limit
   E_SpindleMonit : BOOL ;	//Error spindle monitoring
   E_AxisCtrl : BOOL ;	// Axis control active
   E_MSFine : BOOL ;	// Master/Slave fine
   E_MSCoarse : BOOL ;	// Master/Slave coarse
   E_MSCompContr : BOOL ;	// Master/Slave Compensation controller activ
   E_BitValCtrlOutChang0 : BOOL ;	// Bit value for CTRLOUT_changed 0:  Change setpoint output assignment
   E_BitValCtrlOutChang1 : BOOL ;	// Bit value for CTRLOUT_changed 1:  Change setpoint output assignment
   E_MS : BOOL ;	//Master/ slave active
   f97 : BYTE ;
   E_SyncronFine : BOOL ;	//Synchronism fine
   E_SyncronCoarse : BOOL ;	//Synchronism coarse
   E_ActValCoupling : BOOL ;	//Actual value coupling
   f98_3 : BOOL ;
   E_OverlayMotion : BOOL ;	//Overlaid motion
   E_SWL : BOOL ;	//Speed warning limit reached
   E_AWL : BOOL ;	//Acceleration warning limit reached
   E_EmRetr : BOOL ;	//Emergency retraction active
   E_MasterSp : BOOL ;	//Master spindle
   E_SlaveSp : BOOL ;	//Slave spindle
   f99_2 : BOOL ;
   E_AxisAccel : BOOL ;	//Axis accelerated
   E_Sync : BOOL ;	//Synchronization active
   E_MSR : BOOL ;	//Max speed reached
   E_MAR : BOOL ;	//Max acceleration reached
   E_EmRetrEnabl : BOOL ;	//Emergency retraction enabled
   f100_0 : BOOL ;
   f100_1 : BOOL ;
   E_OscillAxExtRev : BOOL ;	// OscillAxExt Reversal active
   E_StopOscill : BOOL ;	//Oscillation cannot start
   E_ErrorOscill : BOOL ;	//Error during oscillation
   E_SparkOut : BOOL ;	//Spark-out active
   E_OscillMotion : BOOL ;	//Oscillation motion active
   E_Oscill : BOOL ;	//Oscillation active
   f101_0 : BOOL ;
   f101_1 : BOOL ;
   E_GantCOLimit : BOOL ;	//Gantry cut-off limit exceeded
   E_GantWarn : BOOL ;	//Gantry warning limit exceeded
   E_SynRunStart : BOOL ;	//Synchronization run ready to start
   E_GantGroupSyn : BOOL ;	//Gantry grouping is synchronous
   E_GantLeadAxis : BOOL ;	//Gantry leading axis
   E_GantAxis : BOOL ;	//Gantry axis
   f102 : INT ;
   E_AIAxis : ARRAY  [1 .. 31 ] OF BOOL ;	//Active infeed axis[1..31]
   E_SG_SBH : BOOL ;	//Active SG/SBH
   E_ErrLifeS_CRC : BOOL ;	// Error lifesign or CRC-error
   E_ImpdelNCK : BOOL ;	//Delete pulses NCK
   r108_3 : BOOL ;
   r108_4 : BOOL ;
   r108_5 : BOOL ;
   E_SE2 : BOOL ;	//SE 2 active
   E_SRef : BOOL ;	//Axis safely referenced
   E_SN1Plus : BOOL ;	//Actual position > cam position SN1+
   E_SN1Minus : BOOL ;	//Actual position > cam position SN1-
   E_SN2Plus : BOOL ;	//Actual position > cam position SN2+
   E_SN2Minus : BOOL ;	//Actual position > cam position SN2-
   E_SN3Plus : BOOL ;	//Actual position > cam position SN3+
   E_SN3Minus : BOOL ;	//Actual position > cam position SN3-
   E_SN4Plus : BOOL ;	//Actual position > cam position SN4+
   E_SN4Minus : BOOL ;	//Actual position > cam position SN4-
   f110_0 : BOOL ;
   E_SBH : BOOL ;	//Active SBH
   f110_2 : BOOL ;
   E_SG_0 : BOOL ;	//Active SG 0
   E_SG_1 : BOOL ;	//Active SG 1
   E_n_nx : BOOL ;	//n < nx
   f110_6 : BOOL ;
   f110_7 : BOOL ;
   f111_0 : BOOL ;
   f111_1 : BOOL ;
   f111_2 : BOOL ;
   f111_3 : BOOL ;
   E_StopAB : BOOL ;	//Stop A/B active
   E_StopC : BOOL ;	//Stop C active
   E_StopD : BOOL ;	//Stop D active
   E_StopE : BOOL ;	//Stop E active
   E_CamRangeTr1 : BYTE ;	//Cam Range for Cam Track 1
   E_CamRangeTr2 : BYTE ;	//Cam Range for Cam Track 2
   E_CamRangeTr3 : BYTE ;	//Cam Range for Cam Track 3
   E_CamRangeTr4 : BYTE ;	//Cam Range for Cam Track 4
   f116 : BYTE ;
   E_CamTrack1 : BOOL ;	//Cam Track 1
   E_CamTrack2 : BOOL ;	//Cam Track 2
   E_CamTrack3 : BOOL ;	//Cam Track 3
   E_CamTrack4 : BOOL ;	//Cam Track 4
   f117_4 : BOOL ;
   f117_5 : BOOL ;
   f117_6 : BOOL ;
   f117_7 : BOOL ;
   E_CamRangeBitTr1 : ARRAY  [0 .. 14 ] OF //Cam Range Bits for Cam Track 1
   BOOL ;
   E_CamRangeBitTr2 : ARRAY  [0 .. 14 ] OF //Cam Range Bits for Cam Track 2
   BOOL ;
   E_CamRangeBitTr3 : ARRAY  [0 .. 14 ] OF //Cam Range Bits for Cam Track 3
   BOOL ;
   E_CamRangeBitTr4 : ARRAY  [0 .. 14 ] OF //Cam Range Bits for Cam Track 4
   BOOL ;
  END_STRUCT ;	
BEGIN
END_DATA_BLOCK

DATA_BLOCK DB 95
AUTHOR : NUMERIK
FAMILY : _800D
VERSION : 0.0
"GET"
BEGIN
END_DATA_BLOCK

DATA_BLOCK "DB_Ingressi"	// DB 100
VERSION : 0.1
  STRUCT
   Fungo_ConsollePremuto : BOOL ;
   Fungo_CNPremuto : BOOL ;
   Fungo_RobotPremuto : BOOL ;
   RiparoAperto_Robot : BOOL ;
   RiparoAperto_Operatore : BOOL ;
   EXT_Z_Piu : BOOL ;
   EXT_Z_Meno : BOOL ;
   EXT_X_Piu : BOOL ;
   EXT_X_Meno : BOOL ;
   EXT_Y_Piu : BOOL ;
   EXT_Y_Meno : BOOL ;
   PotenzaDriveInserita : BOOL ;
   TermicoLubrificazione : BOOL ;
   TermicoCentralina : BOOL ;
   TermicoRaffr_Centralina : BOOL ;
   TermicoFiltroDrives : BOOL ;
   TermicoCondizArmadio : BOOL ;
   AlimentatorePronto : BOOL ;
   SelBypassExtracorsa : BOOL ;
   Cancello_RobotAperto : BOOL ;
   ErroreTastatoreMarposs : BOOL ;
   BatteriaScaricaMarposs : BOOL ;
   LivelloMaxRefrigerante : BOOL ;
   FlussostatoRefrigEsterno : BOOL ;
   PedaleMandrino1 : BOOL ;
   PedaleMandrino2 : BOOL ;
   PressostatoPortamole : BOOL ;
   PressostatoPinzaPortapez : BOOL ;
   LivMaxCentralinaIdraulic : BOOL ;
   PressPinzaMorsa : BOOL ;
   PressTavolaVerticale : BOOL ;
   PressTavolaOrizzontale : BOOL ;
   RichAperturaPortaOperat : BOOL ;
   RichAperturaPortaRobot : BOOL ;
   RipristinoSicurezze : BOOL ;
   RobotaRiposo : BOOL ;
   RobotProgMode : BOOL ;
   RobotAutoMode : BOOL ;
   PresenzaAria : BOOL ;
   PressostatoLubrificazion : BOOL ;
   LivelloOlioLubrificazion : BOOL ;
   FlussostatoX : BOOL ;
   FlussostatoY : BOOL ;
   FlussostatoZ : BOOL ;
   FlussostatoA : BOOL ;
   FlussostatoB : BOOL ;
   FlussostatoMandrino : BOOL ;
   FlussostatoRettifMola : BOOL ;
   Flussostato8 : BOOL ;
   FcPortapezzoAperto : BOOL ;
   FcPortapezzoChiuso : BOOL ;
   FcMorsaAperta : BOOL ;
   PortapezzoAperto : BOOL ;
   PortapezzoChiuso : BOOL ;
   Sel_MAN_AUTO : BOOL ;
   ConsensoMovimentiManuali : BOOL ;
   FcMorsaChiusa : BOOL ;
   ProtezApertaLatoRob : BOOL ;
   RiparoChiuso_Robot : BOOL ;
   EvRefOlio1_Aperta : BOOL ;
   EvRefOlio1_chiusa : BOOL ;
   EvRefOlio2_Aperta : BOOL ;
   EvRefOlio2_chiusa : BOOL ;
   in63 : BOOL ;
   ModuloARattivo : BOOL ;
   TermicoMotRaffeddamento : BOOL ;
   TermicoPompaTravaso : BOOL ;
   AusiliariInseriti : BOOL ;
   AssiInArrestoSicuro : BOOL ;
   LivMaxVascaInterna : BOOL ;
   LivMinVascaEsterna : BOOL ;
   LivMaxVascaEsterna : BOOL ;
   LivPresenzaOlioLavoraz : BOOL ;
   TermicaPompaTravaso : BOOL ;
   TermicoPompaRefrigerante : BOOL ;
   in75 : BOOL ;
   in76 : BOOL ;
   in77 : BOOL ;
   in78 : BOOL ;
   in79 : BOOL ;
  END_STRUCT ;	
BEGIN
END_DATA_BLOCK

DATA_BLOCK "DB_Uscite"	// DB 101
VERSION : 0.1
  STRUCT
   Lampada_PortaOp_Aperta : BOOL ;
   Lampada_PortaRob_Aperta : BOOL ;
   CicloInAutomatico : BOOL ;
   VentilatoreMandrino : BOOL ;
   MotoreCentralinaIdraulic : BOOL ;
   VentolaCentralina : BOOL ;
   LampadaAllarme : BOOL ;
   LampadaPreallarme : BOOL ;
   LampadaMacchinaPronta : BOOL ;
   LampadaMacchinaAvviata : BOOL ;
   BloccoAsseA : BOOL ;
   ris1 : BOOL ;
   BloccoPinzaAsseA : BOOL ;
   SbloccoPinzaAsseA : BOOL ;
   BloccoAsseB : BOOL ;
   ris2 : BOOL ;
   EV_ApriPortaRobot : BOOL ;
   EV_ChiudiPortaRobot : BOOL ;
   EV_ApriPortaPezzo : BOOL ;
   SoffieriaMandrino : BOOL ;
   SoffieriaAsseA : BOOL ;
   Olio1 : BOOL ;
   Olio2 : BOOL ;
   EsclusioneTastatore : BOOL ;
   EvGeneraleAriaON : BOOL ;
   EvApriMandrino : BOOL ;
   EvChiudiMandrino : BOOL ;
   LampInterventoSicurezze : BOOL ;
   MotoreLubrificazione : BOOL ;
   SbloccoFrenoAsseY : BOOL ;
   EvLubeAsseA : BOOL ;
   EvLubeAsseB : BOOL ;
   SoffieriaPezzo : BOOL ;
   PressurizzRettificaMola : BOOL ;
   PressurizzElettromandrin : BOOL ;
   Ev_SoffieriaPortapezzo : BOOL ;
   Ev_SoffieriaPortamola : BOOL ;
   EV_ApriMorse : BOOL ;
   EV_ChiudiMorse : BOOL ;
   out39 : BOOL ;
   CdoOFF1 : BOOL ;
   CdoOFF3 : BOOL ;
   ArrestaAssiSicuri : BOOL ;
   out43 : BOOL ;
   out44 : BOOL ;
   out45 : BOOL ;
   out46 : BOOL ;
   out47 : BOOL ;
   EvGeneraleRaffeddamento : BOOL ;
   MotoreRaffreddamento : BOOL ;
   MotorePompaTravaso : BOOL ;
   MotoreOlioRefrigerante : BOOL ;
   out52 : BOOL ;
   out53 : BOOL ;
   out54 : BOOL ;
   out55 : BOOL ;
   out56 : BOOL ;
   out57 : BOOL ;
   out58 : BOOL ;
   out59 : BOOL ;
   out60 : BOOL ;
   out61 : BOOL ;
   out62 : BOOL ;
   out63 : BOOL ;
   out64 : BOOL ;
   out65 : BOOL ;
   out66 : BOOL ;
   out67 : BOOL ;
   out68 : BOOL ;
   out69 : BOOL ;
   out70 : BOOL ;
   out71 : BOOL ;
   out72 : BOOL ;
   out73 : BOOL ;
   out74 : BOOL ;
   out75 : BOOL ;
   out76 : BOOL ;
   out77 : BOOL ;
   out78 : BOOL ;
   out79 : BOOL ;
  END_STRUCT ;	
BEGIN
END_DATA_BLOCK

DATA_BLOCK "DB Segnali Macchina"	// DB 102
AUTHOR : Asamec
VERSION : 0.1
  STRUCT
   MacchinaOK : BOOL ;
   MacchinaAccesa : BOOL ;
   PulseMacchinaAccesa : BOOL ;
   MacchinaAccesaRitardato : BOOL ;
   MacchinaInSicurezza : BOOL ;
   RichiestaHold : BOOL ;
   CicloDiCaricoInAuto : BOOL ;
   BloccoLetturaAttivo : BOOL ;
   BloccoAssiAttivo : BOOL ;
   BloccoMandrinoAttivo : BOOL ;
   BloccoAssiEMandrinoAttiv : BOOL ;
   BloccoRipartenzaAttivo : BOOL ;
   MessaggioAttivo : BOOL ;
   MandrinoFermo : BOOL ;
   MacchinaInManuale : BOOL ;
   Comm_OKPress_PP : BOOL ;	//Commutazione Ok pressostato p iza portapezzo
  END_STRUCT ;	
BEGIN
END_DATA_BLOCK

DATA_BLOCK "DB Impostazioni"	// DB 103
VERSION : 0.1
  STRUCT
   TempoLubAsseA : INT ;
   IntervalloLubAsseA : INT ;
   TempoLubAsseB : INT ;
   IntervalloLubAsseB : INT ;
   TempoLubAssi : INT ;
   IntervalloLubAssi : INT ;
   Analog_Min_Pinza_Aperta : INT ;
   Analog_Max_Pinza_Aperta : INT ;
   Analog_Min_Pinza_Chiusa : INT ;
   Analog_Max_Pinza_Chiusa : INT ;
   ContapezziAttuale : INT ;
   NumeroPezziInterv_Tastat : INT ;
   ContapezziTotale : INT ;
   Ris11 : INT ;
   Ris12 : INT ;
   Ris13 : INT ;
   Ris14 : INT ;
   Ris15 : INT ;
   Ris16 : INT ;
   Ris17 : INT ;
   Ris18 : INT ;
   Ris19 : INT ;
   RisReal : REAL ;
   RisReal1 : REAL ;
   RisReal2 : REAL ;
   RisReal3 : REAL ;
   RisReal4 : REAL ;
   RisReal5 : REAL ;
   RisReal6 : REAL ;
   RisReal7 : REAL ;
   RisReal8 : REAL ;
   RisReal9 : REAL ;
   RisReal10 : REAL ;
   RisReal11 : REAL ;
   RisReal12 : REAL ;
   RisReal13 : REAL ;
   RisReal14 : REAL ;
   RisReal15 : REAL ;
   RisReal16 : REAL ;
   RisReal17 : REAL ;
   RisReal18 : REAL ;
   RisReal19 : REAL ;
  END_STRUCT ;	
BEGIN
END_DATA_BLOCK

DATA_BLOCK "PC<>PLC"	// DB 110
VERSION : 0.1
  STRUCT
   Pc_to_Plc : STRUCT
    ConsensoLetturaNrProg : BOOL ;	//Consenso alla esecuzione del programma
    DatoBool_02 : BOOL ;
    DatoBool_03 : BOOL ;
    DatoBool_04 : BOOL ;
    DatoBool_05 : BOOL ;
    DatoBool_06 : BOOL ;
    DatoBool_07 : BOOL ;
    DatoBool_08 : BOOL ;
    DatoBool_09 : BOOL ;
    ApriRiparo : BOOL ;	//Richiesta apertura riparo
    ChiudiRiparo : BOOL ;	//Richiesta chiusura riparo
    ApriMorsetta : BOOL ;	//Richiesta apertura morsa
    ChiudiMorsetta : BOOL ;	//Richiesta chiusura morsa
    DatoBool_014 : BOOL ;
    DatoBool_015 : BOOL ;
    DatoBool_016 : BOOL ;
    DatoBool_017 : BOOL ;
    DatoBool_018 : BOOL ;
    DatoBool_019 : BOOL ;
    DatoBool_020 : BOOL ;
    DatoBool_021 : BOOL ;
    DatoBool_022 : BOOL ;
    DatoBool_023 : BOOL ;
    DatoBool_024 : BOOL ;
    DatoBool_025 : BOOL ;
    DatoBool_026 : BOOL ;
    DatoBool_027 : BOOL ;
    DatoBool_028 : BOOL ;
    DatoBool_029 : BOOL ;
    DatoBool_030 : BOOL ;
    DatoBool_031 : BOOL ;
    DatoBool_032 : BOOL ;
    DatoBool_033 : BOOL ;
    DatoBool_034 : BOOL ;
    DatoBool_035 : BOOL ;
    DatoBool_036 : BOOL ;
    DatoBool_037 : BOOL ;
    DatoBool_038 : BOOL ;
    DatoBool_039 : BOOL ;
    VivoPLC : BOOL ;	//RichiestaControlloComunicazioni
    RichiestaTipo : INT ;	//Richiesta tipo da lavorare
    DAto_02 : INT ;
    DAto_03 : INT ;
    DAto_04 : INT ;
    DAto_05 : INT ;
    DAto_06 : INT ;
    DAto_07 : INT ;
    DAto_08 : INT ;
    DAto_09 : INT ;
    DAto_010 : INT ;
    DAto_011 : INT ;
    DAto_012 : INT ;
    DAto_013 : INT ;
    DAto_014 : INT ;
    DAto_015 : INT ;
    DatoReal_01 : REAL ;
    DatoReal_02 : REAL ;
    DatoReal_03 : REAL ;
    DatoReal_04 : REAL ;
    DatoReal_05 : REAL ;
    DatoReal_06 : REAL ;
    DatoReal_07 : REAL ;
    DatoReal_08 : REAL ;
    DatoReal_09 : REAL ;
    DatoReal_010 : REAL ;
   END_STRUCT ;
   Spare : DINT ;
   Spare1 : DINT ;
   Spare2 : DINT ;
   Spare3 : DINT ;
   Spare4 : DINT ;
   Spare5 : DINT ;
   PLC_to_PC : STRUCT 	//Variabile jolly provvisoria
    NrProgrammaAcquisito : BOOL ;	//Conferma esecuzione programma
    ProntoPerComandi : BOOL ;
    DatoBool_03 : BOOL ;
    DatoBool_04 : BOOL ;
    DatoBool_05 : BOOL ;
    DatoBool_06 : BOOL ;
    DatoBool_07 : BOOL ;
    DatoBool_08 : BOOL ;
    DatoBool_09 : BOOL ;
    RiparoAperto : BOOL ;	//Riparo aperto
    RiparoChiuso : BOOL ;	//Riparo chiuso
    MorsaAperta : BOOL ;	//Morsa aperta
    MorsaChiusa : BOOL ;	//Morsa chiusa
    DatoBool_014 : BOOL ;
    DatoBool_015 : BOOL ;
    DatoBool_016 : BOOL ;
    DatoBool_017 : BOOL ;
    DatoBool_018 : BOOL ;
    DatoBool_019 : BOOL ;
    DatoBool_020 : BOOL ;
    DatoBool_021 : BOOL ;
    DatoBool_022 : BOOL ;
    DatoBool_023 : BOOL ;
    DatoBool_024 : BOOL ;
    DatoBool_025 : BOOL ;
    DatoBool_026 : BOOL ;
    DatoBool_027 : BOOL ;
    DatoBool_028 : BOOL ;
    DatoBool_029 : BOOL ;
    DatoBool_030 : BOOL ;
    DatoBool_031 : BOOL ;
    DatoBool_032 : BOOL ;
    DatoBool_033 : BOOL ;
    DatoBool_034 : BOOL ;
    DatoBool_035 : BOOL ;
    DatoBool_036 : BOOL ;
    DatoBool_037 : BOOL ;
    DatoBool_038 : BOOL ;
    DatoBool_039 : BOOL ;
    PLC_Attivo : BOOL ;	//RispondiControlloComunicazioni
    DAto_01 : INT ;	//Echo Programma accettato
    DAto_02 : INT ;	//Numero Programma richiesto da robot a PCU
    StatiMacchina : INT ;
    DAto_04 : INT ;
    DAto_05 : INT ;
    DAto_06 : INT ;
    DAto_07 : INT ;
    DAto_08 : INT ;
    DAto_09 : INT ;
    DAto_010 : INT ;
    DAto_011 : INT ;
    DAto_012 : INT ;
    DAto_013 : INT ;
    DAto_014 : INT ;
    DAto_015 : INT ;
    DatoReal_01 : REAL ;
    DatoReal_02 : REAL ;
    DatoReal_03 : REAL ;
    DatoReal_04 : REAL ;
    DatoReal_05 : REAL ;
    DatoReal_06 : REAL ;
    DatoReal_07 : REAL ;
    DatoReal_08 : REAL ;
    DatoReal_09 : REAL ;
    DatoReal_010 : REAL ;
   END_STRUCT ;
   ALIVE : TIME ;
  END_STRUCT ;	
BEGIN
END_DATA_BLOCK

DATA_BLOCK "C_K1"	// DB 120
VERSION : 0.0
  STRUCT
   N_SEMA_measPos11_5 : STRUCT
    SYNTAX_ID : BYTE  := B#16#82;
    Area_Unit : BYTE  := B#16#1;
    Column : WORD  := W#16#5;
    Line : WORD  := W#16#1;
    BlockType : BYTE  := B#16#71;
    NumOfLine : BYTE  := B#16#1;
    DataType : BYTE  := B#16#F;
    Length : BYTE  := B#16#8;
   END_STRUCT ;
  END_STRUCT ;	
BEGIN
   N_SEMA_measPos11_5.SYNTAX_ID := B#16#82;
   N_SEMA_measPos11_5.Area_Unit := B#16#1;
   N_SEMA_measPos11_5.Column := W#16#5;
   N_SEMA_measPos11_5.Line := W#16#1;
   N_SEMA_measPos11_5.BlockType := B#16#71;
   N_SEMA_measPos11_5.NumOfLine := B#16#1;
   N_SEMA_measPos11_5.DataType := B#16#F;
   N_SEMA_measPos11_5.Length := B#16#8;
END_DATA_BLOCK

DATA_BLOCK "DB Ist-Analigiche"	// DB 200
VERSION : 0.0
"FB Analogiche"
BEGIN
END_DATA_BLOCK

ORGANIZATION_BLOCK "OB 1"	// OB 1
VERSION : 1.0
VAR_TEMP
  OB1_EV_CLASS : BYTE ;
  OB1_SCAN_1 : BYTE ;
  OB1_PRIORITY : BYTE ;
  OB1_OB_NUMBR : BYTE ;
  OB1_RESERVED_1 : BYTE ;
  OB1_RESERVED_2 : BYTE ;
  OB1_PREV_CYCLE : INT ;
  OB1_MIN_CYCLE : INT ;
  OB1_MAX_CYCLE : INT ;
  OB1_DATE_TIME : DATE_AND_TIME ;
END_VAR
BEGIN
NETWORK
TITLE =
      CALL  "GP_HP";
//Insert User program from here
      CALL  "AL_MSG" (
           $1                       := TRUE,
           $2                       := TRUE);
NETWORK
TITLE = Pulsante lubrificazione
      A     I 5.4;
      R     I 5.4;
      =     "M35.1";
NETWORK
TITLE =
      CALL  "FC Ingressi";
      CALL  "FC Generali";
      CALL  "FC Idraulica";
      CALL  "FC Assi";
      CALL  "FC Refrigerante";
      CALL  "FC Mandrino";
      CALL  "FC Ausiliari";
      CALL  "FC Lubrificazioni";
      CALL  "FC Allarmi";
      CALL  "FC Tastatura";
NETWORK
TITLE = Safety
      A     "DB Segnali Macchina".MacchinaAccesa;
      =     "DB_Uscite".ArrestaAssiSicuri;
NETWORK
TITLE =
      CALL  "FC Uscite";
NETWORK
TITLE =
      CALL  "FC ComPCPlc";
END_ORGANIZATION_BLOCK

ORGANIZATION_BLOCK OB 40
VERSION : 1.0
VAR_TEMP
  OB40_EV_CLASS : BYTE ;
  OB40_STRT_INF : BYTE ;
  OB40_PRIORITY : BYTE ;
  OB40_OB_NUMBR : BYTE ;
  OB40_RESERVED_1 : BYTE ;
  OB40_MDL_ID : BYTE ;
  OB40_MDL_ADDR : INT ;
  OB40_POINT_ADDR : DWORD ;
  OB40_DATE_TIME : DATE_AND_TIME ;	//data for the Basic program
  GP_IRFromNCK : BOOL ;	//Interrupt from NCK
  GP_TM : BOOL ;	//Toolmanagment
  GP_InPosition : ARRAY  [1 .. 31 ] OF BOOL ;	//InPos Signal from FC15,16,18
  GP_AuxFunction : ARRAY  [1 .. 10 ] OF BOOL ;	//auxiliary functions
  GP_FMBlock : ARRAY  [1 .. 10 ] OF BOOL ;	//not used
//Insert User-data from here
END_VAR
BEGIN
NETWORK
TITLE =
      CALL  "GP_PRAL";
//Insert User program from here
END_ORGANIZATION_BLOCK

ORGANIZATION_BLOCK OB 82
TITLE = "I/O Point Fault"
VERSION : 1.0
VAR_TEMP
  OB82_EV_CLASS : BYTE ;	//16#39, Event class 3, Entering event state, Internal fault event
  OB82_FLT_ID : BYTE ;	//16#XX, Fault identifcation code
  OB82_PRIORITY : BYTE ;	//Priority of OB Execution
  OB82_OB_NUMBR : BYTE ;	//82 (Organization block 82, OB82)
  OB82_RESERVED_1 : BYTE ;	//Reserved for system
  OB82_IO_FLAG : BYTE ;	//Input (01010100), Output (01010101)
  OB82_MDL_ADDR : WORD ;	//Base address of module with fault
  OB82_MDL_DEFECT : BOOL ;	//Module defective
  OB82_INT_FAULT : BOOL ;	//Internal fault
  OB82_EXT_FAULT : BOOL ;	//External fault
  OB82_PNT_INFO : BOOL ;	//Point information
  OB82_EXT_VOLTAGE : BOOL ;	//External voltage low
  OB82_FLD_CONNCTR : BOOL ;	//Field wiring connector missing
  OB82_NO_CONFIG : BOOL ;	//Module has no configuration data
  OB82_CONFIG_ERR : BOOL ;	//Module has configuration error
  OB82_MDL_TYPE : BYTE ;	//Type of module
  OB82_SUB_MDL_ERR : BOOL ;	//Sub-Module is missing or has error
  OB82_COMM_FAULT : BOOL ;	//Communication fault
  OB82_MDL_STOP : BOOL ;	//Module is stopped
  OB82_WTCH_DOG_FLT : BOOL ;	//Watch dog timer stopped module
  OB82_INT_PS_FLT : BOOL ;	//Internal power supply fault
  OB82_PRIM_BATT_FLT : BOOL ;	//Primary battery is in fault
  OB82_BCKUP_BATT_FLT : BOOL ;	//Backup battery is in fault
  OB82_RESERVED_2 : BOOL ;	//Reserved for system
  OB82_RACK_FLT : BOOL ;	//Rack fault, only for bus interface module
  OB82_PROC_FLT : BOOL ;	//Processor fault
  OB82_EPROM_FLT : BOOL ;	//EPROM fault
  OB82_RAM_FLT : BOOL ;	//RAM fault
  OB82_ADU_FLT : BOOL ;	//ADU fault
  OB82_FUSE_FLT : BOOL ;	//Fuse fault
  OB82_HW_INTR_FLT : BOOL ;	//Hardware interupt input in fault
  OB82_RESERVED_3 : BOOL ;	//Reserved for system
  OB82_DATE_TIME : DATE_AND_TIME ;	//Date and time OB82 started
END_VAR
BEGIN
NETWORK
TITLE = Detailed Diagnosis in OB82 (interrupt)
      CALL  "GP_DIAG" (
           $1                       := TRUE);
END_ORGANIZATION_BLOCK

ORGANIZATION_BLOCK OB 86
TITLE = "Loss Of Rack Fault"
VERSION : 1.0
VAR_TEMP
  OB86_EV_CLASS : BYTE ;	//16#38/39 Event class 3
  OB86_FLT_ID : BYTE ;	//16#C1/C4/C5, Fault identifcation code
  OB86_PRIORITY : BYTE ;	//Priority of OB Execution
  OB86_OB_NUMBR : BYTE ;	//86 (Organization block 86, OB86)
  OB86_RESERVED_1 : BYTE ;	//Reserved for system
  OB86_RESERVED_2 : BYTE ;	//Reserved for system
  OB86_MDL_ADDR : WORD ;	//Base address of IM module in rack with fault
  OB86_RACKS_FLTD : ARRAY  [0 .. 31 ] OF BOOL ;	//Racks in fault
  OB86_DATE_TIME : DATE_AND_TIME ;	//Date and time OB86 started
END_VAR
BEGIN
NETWORK
TITLE = Detailed Diagnosis in OB86 (interrupt)
      CALL  "GP_DIAG" (
           $1                       := TRUE);
END_ORGANIZATION_BLOCK

ORGANIZATION_BLOCK OB 100
VERSION : 1.0
VAR_TEMP
  OB100_EV_CLASS : BYTE ;
  OB100_STRTUP : BYTE ;
  OB100_PRIORITY : BYTE ;
  OB100_OB_NUMBR : BYTE ;
  OB100_RESERVED_1 : BYTE ;
  OB100_RESERVED_2 : BYTE ;
  OB100_STOP : WORD ;
  OB100_RESERVED_3 : WORD ;
  OB100_RESERVED_4 : WORD ;
  OB100_DATE_TIME : DATE_AND_TIME ;
END_VAR
BEGIN
NETWORK
TITLE =
      CALL  "RUN_UP" , "gp_par" (
           DIW 0                    := 1,
           DIW 2                    := 0,
           DID 4                    := P#I 0.0,
           DIW 8                    := 0,
           DID 10                   := P#Q 0.0,
           DIW 14                   := 0,
           DID 16                   := P#Q 8.0,
           DIW 20                   := 0,
           DID 22                   := P#Q 12.0,
           DIW 26                   := 192,
           DIB 63                   := B#16#55,
           DIX 116.0                := TRUE);
//Insert User program from here
END_ORGANIZATION_BLOCK

SYMBOL_TABLE
"DB Allarmi"	DB 2	DB 2
"gp_par"	DB 7	FB 1	// Parameters for Baseprogram
"DB SegnaliMacchina"	DB 9	DB 9
"NC"	DB 10	UDT 10
"BAG"	DB 11	UDT 11
"PI"	DB 16	DB 16	// Datainterface PI-Services
"SPL"	DB 18	DB 18	// SPL dataarea
"MMC"	DB 19	UDT 19
"Chan1"	DB 21	UDT 21
"Asse_X"	DB 31	UDT 31
"Asse_Y"	DB 32	UDT 31
"Asse_Z"	DB 33	UDT 31
"Asse_A"	DB 34	UDT 31
"Asse_B"	DB 35	UDT 31
"Asse_Mandrino"	DB 36	UDT 31
"Asse_Mag"	DB 37	UDT 31
"DB Ingressi"	DB 100	DB 100
"DB Uscite"	DB 101	DB 101
"DB Ist-Analigiche"	DB 200	FB 200
"RUN_UP"	FB 1	FB 1	// Startup Baseprogram
"GET"	FB 2	FB 2	// read NC Variable
"PUT"	FB 3	FB 3	// write NC Variable
"PI_SERV"	FB 4	FB 4	// PI-Services 1
"GETGUD"	FB 5	FB 5	// read GUD-Variable
"PI_SERV2"	FB 7	FB 7	// PI-Services 2
"M2N"	FB 9	FB 9	// Several OPs/NCUs
"SI_Relais"	FB 10	FB 10	// Safety Integrated: Relais
"SI_BrakeTest"	FB 11	FB 11	// Safety Integrated: Brake Test
"Diagnose"	FB 29	FB 29	// Signal recorder and data trigger diagnostics
"Lettura_Gud"	FB 100	FB 100
"FB Analogiche"	FB 200	FB 200
"GP_HP"	FC 2	FC 2	// cyclic Baseprogram
"GP_PRAL"	FC 3	FC 3	// alarmtriggered Baseprogram
"GP_DIAG"	FC 5	FC 5	// Diagnosis alarm and Modul failure
"TM_REV"	FC 7	FC 7	// Transfer for Revolverchange
"TM_TRANS"	FC 8	FC 8	// Transfer for Toolmanagment
"ASUP"	FC 9	FC 9	// asynchronous Subprograms
"AL_MSG"	FC 10	FC 10	// Alarms & Messages
"BHGDisp"	FC 13	FC 13	// Displaycontrol for Handheld Unit
"YDelta"	FC 17	FC 17	// Y / Delta Control
"SpinCtrl"	FC 18	FC 18	// Spindlecontrol / Part-, Positioning-axis
"MCP_IFM"	FC 19	FC 19	// MCP-Signals to Interface, Variant M
"Transfer"	FC 21	FC 21	// Quick Datachannel
"TM_DIR"	FC 22	FC 22	// Directioncontrol for Toolmanagment Mag.
"MCP_IFM2"	FC 24	FC 24	// MCP-Signals to Interface, Variant small
"MCP_IFT"	FC 25	FC 25	// MCP-Signals to Interface, Variant T
"HPU_MCP"	FC 26	FC 26	// MCP-Signals of PHG to Interface
"FC Analogiche"	FC 97	FC 97
"FC DecodM"	FC 98	FC 98	// DECODIFICA FUNZIONI WORD-BIT
"FC Gestione Allarmi"	FC 99	FC 99
"FC Generali"	FC 100	FC 100
"FC Ingressi/Uscite"	FC 102	FC 102
"FC Allarmi"	FC 103	FC 103
"FC Sicurezze"	FC 104	FC 104
"FC Mandrino"	FC 105	FC 105
"FC Refrigerante"	FC 106	FC 106
"SCALE"	FC 200	FC 200	// Scaling Values
"Pulsantiera.Reset"	I 3.7	BOOL
"Log1"	M 0.0	BOOL	// Bit sempre a 1
"Pulsantiera.FeedHold"	M 0.2	BOOL
"Pulsatiera.SpindleHold"	M 0.3	BOOL
"Occhio"	M 0.5	BOOL
"MessainServizio"	M 0.7	BOOL
"Funzione M Attiva"	M 1.2	BOOL
"M10.0"	M 10.0	BOOL
"M10.1"	M 10.1	BOOL
"M10.3"	M 10.3	BOOL
"M10.4"	M 10.4	BOOL
"FC_Mandrino_Aperto"	M 100.0	BOOL
"FC_Mandrino_Chiuso"	M 100.1	BOOL
"M100.2"	M 100.2	BOOL
"M100.3"	M 100.3	BOOL
"M100.4"	M 100.4	BOOL
"M100.5"	M 100.5	BOOL
"M200.0"	M 200.0	BOOL
"M00"	M 220.0	BOOL	// Stop Programma
"M01"	M 220.1	BOOL	// Stop Programma Opzionale
"M02"	M 220.2	BOOL
"M03"	M 220.3	BOOL	// Rotazione Mandrino Oraria
"M04"	M 220.4	BOOL	// Rotazione Mandrino Antioraria
"M05"	M 220.5	BOOL	// Stop Mandrino
"M06"	M 220.6	BOOL
"M07"	M 220.7	BOOL	// Attiva refrigerante 1
"M08"	M 221.0	BOOL	// Attiva refrigerante 2
"M09"	M 221.1	BOOL	// Stop Refrigerante
"M10"	M 221.2	BOOL
"M11"	M 221.3	BOOL
"M12"	M 221.4	BOOL
"M13"	M 221.5	BOOL
"M14"	M 221.6	BOOL
"M15"	M 221.7	BOOL
"M16"	M 222.0	BOOL
"M17"	M 222.1	BOOL	// Fine Sottoprogramma
"M18"	M 222.2	BOOL
"M19"	M 222.3	BOOL
"M20"	M 222.4	BOOL	// Sblocca Utensile
"M21"	M 222.5	BOOL	// Blocca Utensile
"M22"	M 222.6	BOOL
"M23"	M 222.7	BOOL
"M25"	M 223.1	BOOL
"M26"	M 223.2	BOOL
"M27"	M 223.3	BOOL
"M28"	M 223.4	BOOL
"M29"	M 223.5	BOOL
"M30"	M 223.6	BOOL	// Reset
"M31"	M 223.7	BOOL
"M32"	M 224.0	BOOL
"M33"	M 224.1	BOOL
"M34"	M 224.2	BOOL
"M35"	M 224.3	BOOL
"M36"	M 224.4	BOOL
"M37"	M 224.5	BOOL
"M38"	M 224.6	BOOL
"M39"	M 224.7	BOOL
"M40"	M 225.0	BOOL
"M41"	M 225.1	BOOL
"M42"	M 225.2	BOOL
"M43"	M 225.3	BOOL
"M44"	M 225.4	BOOL
"M45"	M 225.5	BOOL
"M46"	M 225.6	BOOL
"M47"	M 225.7	BOOL
"M48"	M 226.0	BOOL
"M49"	M 226.1	BOOL
"M50"	M 226.2	BOOL
"M51"	M 226.3	BOOL
"M52"	M 226.4	BOOL
"M53"	M 226.5	BOOL
"M54"	M 226.6	BOOL
"M55"	M 226.7	BOOL
"M56"	M 227.0	BOOL
"M57"	M 227.1	BOOL
"M58"	M 227.2	BOOL
"M59"	M 227.3	BOOL
"M61"	M 227.5	BOOL
"M62"	M 227.6	BOOL
"M63"	M 227.7	BOOL
"M64"	M 228.0	BOOL
"M65"	M 228.1	BOOL
"M66"	M 228.2	BOOL
"M67"	M 228.3	BOOL
"M68"	M 228.4	BOOL
"M69"	M 228.5	BOOL
"M70"	M 228.6	BOOL
"M71"	M 228.7	BOOL
"M72"	M 229.0	BOOL	// Apertura Riparo
"M73"	M 229.1	BOOL	// Chiusura Riparo
"M74"	M 229.2	BOOL
"M75"	M 229.3	BOOL
"M76"	M 229.4	BOOL
"M77"	M 229.5	BOOL
"M78"	M 229.6	BOOL
"M79"	M 229.7	BOOL
"M80"	M 230.0	BOOL
"M81"	M 230.1	BOOL
"M82"	M 230.2	BOOL
"M83"	M 230.3	BOOL
"M84"	M 230.4	BOOL
"M85"	M 230.5	BOOL
"M86"	M 230.6	BOOL
"M87"	M 230.7	BOOL
"M88"	M 231.0	BOOL
"M89"	M 231.1	BOOL
"M90"	M 231.2	BOOL
"M91"	M 231.3	BOOL
"M92"	M 231.4	BOOL
"M93"	M 231.5	BOOL
"M94"	M 231.6	BOOL
"M95"	M 231.7	BOOL
"M96"	M 232.0	BOOL
"M97"	M 232.1	BOOL
"M98"	M 232.2	BOOL
"M99"	M 232.3	BOOL
"M100"	M 232.4	BOOL
"Clock_200ms"	M 255.3	BOOL
"OB 1"	OB 1	OB 1
"TON"	SFB 4	SFB 4	// Generate an On Delay
"ALARM_SQ"	SFC 17	SFC 17	// Generate Block-Related Messages with Acknowledgment
"FILL"	SFC 21	SFC 21	// Initialize a Memory Area
"TIME_TCK"	SFC 64	SFC 64	// Read the System Time
"T1"	T 1	TIMER
"T2"	T 2	TIMER
"T3"	T 3	TIMER
"T4"	T 4	TIMER
"T5"	T 5	TIMER
"T6"	T 6	TIMER
END_SYMBOL_TABLE

TYPE UDT 2
VERSION : 0.0
  STRUCT
   C1 : STRUCT 	//From Channel 1
    FDD_5100xx : ARRAY  [0 .. 15 ] OF //Feed disable A.no.51000-510015
    BOOL ;
    FDD_RID_5101xx : ARRAY  [0 .. 31 ] OF //Feed and read-in disable A.no.510100-510131
    BOOL ;
    RID_5102xx : ARRAY  [0 .. 31 ] OF //Read-in disable A.no.510200-510231
    BOOL ;
    NCSD_5103xx : ARRAY  [0 .. 15 ] OF //NC start disable A.no.510300-510315
    BOOL ;
    FdStop_1_5111xx : ARRAY  [0 .. 15 ] OF //Feed stop GEOaxis 1 A.no.511100-511115
    BOOL ;
    FdStop_2_5112xx : ARRAY  [0 .. 15 ] OF //Feed stop GEOaxis 2 A.no.511200-511215
    BOOL ;
    FdStop_3_5113xx : ARRAY  [0 .. 15 ] OF //Feed stop GEOaxis 3 A.no.511300-511315
    BOOL ;
   END_STRUCT ;
   C2 : STRUCT 	//From Channel 2
    FDD_5200xx : ARRAY  [0 .. 15 ] OF //Feed disable A.no.520000-520015
    BOOL ;
    FDD_RID_5201xx : ARRAY  [0 .. 31 ] OF //Feed and read-in disable A.no.520100-520131
    BOOL ;
    RID_5202xx : ARRAY  [0 .. 31 ] OF //Read-in disable A.no.520200-520231
    BOOL ;
    NCSD_5203xx : ARRAY  [0 .. 15 ] OF //NC start disable A.no.520300-520315
    BOOL ;
    FdStop_1_5211xx : ARRAY  [0 .. 15 ] OF //Feed stop GEOaxis 1 A.no.521100-521115
    BOOL ;
    FdStop_2_5212xx : ARRAY  [0 .. 15 ] OF //Feed stop GEOaxis 2 A.no.521200-521215
    BOOL ;
    FdStop_3_5213xx : ARRAY  [0 .. 15 ] OF //Feed stop GEOaxis 3 A.no.521300-521315
    BOOL ;
   END_STRUCT ;
   C3 : STRUCT 	//From Channel 3
    FDD_5300xx : ARRAY  [0 .. 15 ] OF //Feed disable A.no.530000-530015
    BOOL ;
    FDD_RID_5301xx : ARRAY  [0 .. 31 ] OF //Feed and read-in disable A.no.530100-530131
    BOOL ;
    RID_5302xx : ARRAY  [0 .. 31 ] OF //Read-in disable A.no.530200-530231
    BOOL ;
    NCSD_5303xx : ARRAY  [0 .. 15 ] OF //NC start disable A.no.530300-530315
    BOOL ;
    FdStop_1_5311xx : ARRAY  [0 .. 15 ] OF //Feed stop GEOaxis 1 A.no.531100-531115
    BOOL ;
    FdStop_2_5312xx : ARRAY  [0 .. 15 ] OF //Feed stop GEOaxis 2 A.no.531200-531215
    BOOL ;
    FdStop_3_5313xx : ARRAY  [0 .. 15 ] OF //Feed stop GEOaxis 3 A.no.531300-531315
    BOOL ;
   END_STRUCT ;
   C4 : STRUCT 	//From Channel 4
    FDD_5400xx : ARRAY  [0 .. 15 ] OF //Feed disable A.no.540000-540015
    BOOL ;
    FDD_RID_5401xx : ARRAY  [0 .. 31 ] OF //Feed and read-in disable A.no.540100-540131
    BOOL ;
    RID_5402xx : ARRAY  [0 .. 31 ] OF //Read-in disable A.no.540200-540231
    BOOL ;
    NCSD_5403xx : ARRAY  [0 .. 15 ] OF //NC start disable A.no.540300-540315
    BOOL ;
    FdStop_1_5411xx : ARRAY  [0 .. 15 ] OF //Feed stop GEOaxis 1 A.no.541100-541115
    BOOL ;
    FdStop_2_5412xx : ARRAY  [0 .. 15 ] OF //Feed stop GEOaxis 2 A.no.541200-541215
    BOOL ;
    FdStop_3_5413xx : ARRAY  [0 .. 15 ] OF //Feed stop GEOaxis 3 A.no.541300-541315
    BOOL ;
   END_STRUCT ;
   C5 : STRUCT 	//From Channel 5
    FDD_5500xx : ARRAY  [0 .. 15 ] OF //Feed disable A.no.550000-550015
    BOOL ;
    FDD_RID_5501xx : ARRAY  [0 .. 31 ] OF //Feed and read-in disable A.no.550100-550131
    BOOL ;
    RID_5502xx : ARRAY  [0 .. 31 ] OF //Read-in disable A.no.550200-550231
    BOOL ;
    NCSD_5503xx : ARRAY  [0 .. 15 ] OF //NC start disable A.no.550300-550315
    BOOL ;
    FdStop_1_5511xx : ARRAY  [0 .. 15 ] OF //Feed stop GEOaxis 1 A.no.551100-551115
    BOOL ;
    FdStop_2_5512xx : ARRAY  [0 .. 15 ] OF //Feed stop GEOaxis 2 A.no.551200-551215
    BOOL ;
    FdStop_3_5513xx : ARRAY  [0 .. 15 ] OF //Feed stop GEOaxis 3 A.no.551300-551315
    BOOL ;
   END_STRUCT ;
   C6 : STRUCT 	//From Channel 6
    FDD_5600xx : ARRAY  [0 .. 15 ] OF //Feed disable A.no.560000-560015
    BOOL ;
    FDD_RID_5601xx : ARRAY  [0 .. 31 ] OF //Feed and read-in disable A.no.560100-560131
    BOOL ;
    RID_5602xx : ARRAY  [0 .. 31 ] OF //Read-in disable A.no.560200-560231
    BOOL ;
    NCSD_5603xx : ARRAY  [0 .. 15 ] OF //NC start disable A.no.560300-560315
    BOOL ;
    FdStop_1_5611xx : ARRAY  [0 .. 15 ] OF //Feed stop GEOaxis 1 A.no.561100-561115
    BOOL ;
    FdStop_2_5612xx : ARRAY  [0 .. 15 ] OF //Feed stop GEOaxis 2 A.no.561200-561215
    BOOL ;
    FdStop_3_5613xx : ARRAY  [0 .. 15 ] OF //Feed stop GEOaxis 3 A.no.561300-561315
    BOOL ;
   END_STRUCT ;
   C7 : STRUCT 	//From Channel 7
    FDD_5700xx : ARRAY  [0 .. 15 ] OF //Feed disable A.no.570000-570015
    BOOL ;
    FDD_RID_5701xx : ARRAY  [0 .. 31 ] OF //Feed and read-in disable A.no.570100-570131
    BOOL ;
    RID_5702xx : ARRAY  [0 .. 31 ] OF //Read-in disable A.no.570200-570231
    BOOL ;
    NCSD_5703xx : ARRAY  [0 .. 15 ] OF //NC start disable A.no.570300-570315
    BOOL ;
    FdStop_1_5711xx : ARRAY  [0 .. 15 ] OF //Feed stop GEOaxis 1 A.no.571100-511115
    BOOL ;
    FdStop_2_5712xx : ARRAY  [0 .. 15 ] OF //Feed stop GEOaxis 2 A.no.571200-511215
    BOOL ;
    FdStop_3_5713xx : ARRAY  [0 .. 15 ] OF //Feed stop GEOaxis 3 A.no.571300-511315
    BOOL ;
   END_STRUCT ;
   C8 : STRUCT 	//From Channel 8
    FDD_5800xx : ARRAY  [0 .. 15 ] OF //Feed disable A.no.580000-580015
    BOOL ;
    FDD_RID_5801xx : ARRAY  [0 .. 31 ] OF //Feed and read-in disable A.no.580100-510131
    BOOL ;
    RID_5802xx : ARRAY  [0 .. 31 ] OF //Read-in disable A.no.580200-580231
    BOOL ;
    NCSD_5803xx : ARRAY  [0 .. 15 ] OF //NC start disable A.no.580300-580315
    BOOL ;
    FdStop_1_5811xx : ARRAY  [0 .. 15 ] OF //Feed stop GEOaxis 1 A.no.581100-511115
    BOOL ;
    FdStop_2_5812xx : ARRAY  [0 .. 15 ] OF //Feed stop GEOaxis 2 A.no.581200-511215
    BOOL ;
    FdStop_3_5813xx : ARRAY  [0 .. 15 ] OF //Feed stop GEOaxis 3 A.no.581300-511315
    BOOL ;
   END_STRUCT ;
   _1FdStop6001xx : ARRAY  [0 .. 15 ] OF //Feed stop axis/spindle 1
   BOOL ;
   _2FdStop6002xx : ARRAY  [0 .. 15 ] OF //Feed stop axis/spindle 2
   BOOL ;
   _3FdStop6003xx : ARRAY  [0 .. 15 ] OF //Feed stop axis/spindle 3
   BOOL ;
   _4FdStop6004xx : ARRAY  [0 .. 15 ] OF //Feed stop axis/spindle 4
   BOOL ;
   _5FdStop6005xx : ARRAY  [0 .. 15 ] OF //Feed stop axis/spindle 5
   BOOL ;
   _6FdStop6006xx : ARRAY  [0 .. 15 ] OF //Feed stop axis/spindle 6
   BOOL ;
   _7FdStop6007xx : ARRAY  [0 .. 15 ] OF //Feed stop axis/spindle 7
   BOOL ;
   _8FdStop6008xx : ARRAY  [0 .. 15 ] OF //Feed stop axis/spindle 8
   BOOL ;
   _9FdStop6009xx : ARRAY  [0 .. 15 ] OF //Feed stop axis/spindle 9
   BOOL ;
   _10FdStop6010xx : ARRAY  [0 .. 15 ] OF //Feed stop axis/spindle 10
   BOOL ;
   _11FdStop6011xx : ARRAY  [0 .. 15 ] OF //Feed stop axis/spindle 11
   BOOL ;
   _12FdStop6012xx : ARRAY  [0 .. 15 ] OF //Feed stop axis/spindle 12
   BOOL ;
   _13FdStop6013xx : ARRAY  [0 .. 15 ] OF //Feed stop axis/spindle 13
   BOOL ;
   _14FdStop6014xx : ARRAY  [0 .. 15 ] OF //Feed stop axis/spindle 14
   BOOL ;
   _15FdStop6015xx : ARRAY  [0 .. 15 ] OF //Feed stop axis/spindle 15
   BOOL ;
   _16FdStop6016xx : ARRAY  [0 .. 15 ] OF //Feed stop axis/spindle 16
   BOOL ;
   _17FdStop6017xx : ARRAY  [0 .. 15 ] OF //Feed stop axis/spindle 17
   BOOL ;
   _18FdStop6018xx : ARRAY  [0 .. 15 ] OF //Feed stop axis/spindle 18
   BOOL ;
   A7000xx : ARRAY  [0 .. 63 ] OF //Alarm 700000-700063 (user area 0)
   BOOL ;
   A7001xx : ARRAY  [0 .. 63 ] OF //Alarm 700100-700163 (user area 1)
   BOOL ;
   A7002xx : ARRAY  [0 .. 63 ] OF //Alarm 700200-700263 (user area 2)
   BOOL ;
   A7003xx : ARRAY  [0 .. 63 ] OF //Alarm 700300-700363 (user area 3)
   BOOL ;
   A7004xx : ARRAY  [0 .. 63 ] OF //Alarm 700400-700463 (user area 4)
   BOOL ;
   A7005xx : ARRAY  [0 .. 63 ] OF //Alarm 700500-700563 (user area 5
   BOOL ;
   A7006xx : ARRAY  [0 .. 63 ] OF //Alarm 700600-700663 (user area 6)
   BOOL ;
   A7007xx : ARRAY  [0 .. 63 ] OF //Alarm 700700-700763 (user area 7)
   BOOL ;
   A7008xx : ARRAY  [0 .. 63 ] OF //Alarm 700800-700863 (user area 8)
   BOOL ;
   A7009xx : ARRAY  [0 .. 63 ] OF //Alarm 700900-700963 (user area 9)
   BOOL ;
  END_STRUCT ;	
END_TYPE

TYPE UDT 10
VERSION : 0.0
  STRUCT
   A_Disabl_Inp1 : BOOL ;	//Disable digi. NCK input 1
   A_Disabl_Inp2 : BOOL ;	//Disable digi. NCK input 2
   A_Disabl_Inp3 : BOOL ;	//Disable digi. NCK input 3
   A_Disabl_Inp4 : BOOL ;	//Disable digi. NCK input 4
   A_Disabl_Inp5 : BOOL ;	//Disable digi. NCK input 5
   A_Disabl_Inp6 : BOOL ;	//Disable digi. NCK input 6
   A_Disabl_Inp7 : BOOL ;	//Disable digi. NCK input 7
   A_Disabl_Inp8 : BOOL ;	//Disable digi. NCK input 8
   A_Set_Inp1 : BOOL ;	//Set digi. NCK input 1
   A_Set_Inp2 : BOOL ;	//Set digi. NCK input 2
   A_Set_Inp3 : BOOL ;	//Set digi. NCK input 3
   A_Set_Inp4 : BOOL ;	//Set digi. NCK input 4
   A_Set_Inp5 : BOOL ;	//Set digi. NCK input 5
   A_Set_Inp6 : BOOL ;	//Set digi. NCK input 6
   A_Set_Inp7 : BOOL ;	//Set digi. NCK input 7
   A_Set_Inp8 : BOOL ;	//Set digi. NCK input 8
   f0_f15 : ARRAY  [0 .. 15 ] OF BOOL ;	//Reserved
   A_Disabl_Out1 : BOOL ;	//Disable digi. NCK output 1
   A_Disabl_Out2 : BOOL ;	//Disable digi. NCK output 2
   A_Disabl_Out3 : BOOL ;	//Disable digi. NCK output 3
   A_Disabl_Out4 : BOOL ;	//Disable digi. NCK output 4
   A_Disabl_Out5 : BOOL ;	//Disable digi. NCK output 5
   A_Disabl_Out6 : BOOL ;	//Disable digi. NCK output 6
   A_Disabl_Out7 : BOOL ;	//Disable digi. NCK output 7
   A_Disabl_Out8 : BOOL ;	//Disable digi. NCK output 8
   A_OvMask_Out1 : BOOL ;	//Overwrite mask of digi. output 1
   A_OvMask_Out2 : BOOL ;	//Overwrite mask of digi. output 2
   A_OvMask_Out3 : BOOL ;	//Overwrite mask of digi. output 3
   A_OvMask_Out4 : BOOL ;	//Overwrite mask of digi. output 4
   A_OvMask_Out5 : BOOL ;	//Overwrite mask of digi. output 5
   A_OvMask_Out6 : BOOL ;	//Overwrite mask of digi. output 6
   A_OvMask_Out7 : BOOL ;	//Overwrite mask of digi. output 7
   A_OvMask_Out8 : BOOL ;	//Overwrite mask of digi. output 8
   A_Set_Out1 : BOOL ;	//Set digi. NCK output 1
   A_Set_Out2 : BOOL ;	//Set digi. NCK output 2
   A_Set_Out3 : BOOL ;	//Set digi. NCK output 3
   A_Set_Out4 : BOOL ;	//Set digi. NCK output 4
   A_Set_Out5 : BOOL ;	//Set digi. NCK output 5
   A_Set_Out6 : BOOL ;	//Set digi. NCK output 6
   A_Set_Out7 : BOOL ;	//Set digi. NCK output 7
   A_Set_Out8 : BOOL ;	//Set digi. NCK output 8
   A_InMask_Out1 : BOOL ;	//Input mask of digi. output 1
   A_InMask_Out2 : BOOL ;	//Input mask of digi. output 2
   A_InMask_Out3 : BOOL ;	//Input mask of digi. output 3
   A_InMask_Out4 : BOOL ;	//Input mask of digi. output 4
   A_InMask_Out5 : BOOL ;	//Input mask of digi. output 5
   A_InMask_Out6 : BOOL ;	//Input mask of digi. output 6
   A_InMask_Out7 : BOOL ;	//Input mask of digi. output 7
   A_InMask_Out8 : BOOL ;	//Input mask of digi. output 8
   MCP1AxisTbl : ARRAY  [1 .. 22 ] OF BYTE  := B#16#1, B#16#2, B#16#3, B#16#4, B#16#5, B#16#6, B#16#7, B#16#8, B#16#9, B#16#A, B#16#B, B#16#C;	//Axis No. Table MCP1
   MCP1MaxAxis : WORD ;	//max. of Axisno, must be smaller or equal gp_par.MaxAxis
   MCP2AxisTbl : ARRAY  [1 .. 22 ] OF BYTE  := B#16#1, B#16#2, B#16#3, B#16#4, B#16#5, B#16#6, B#16#7, B#16#8, B#16#9, B#16#A, B#16#B, B#16#C;	//Axis No. Table MCP2
   MCP2MaxAxis : WORD ;	//max. of Axisno, must be smaller or equal gp_par.MaxAxis
   f56_0 : BOOL ;
   A_EMERGENCY : BOOL ;	//Emergency stop
   A_EMERGENCY_Ackn : BOOL ;	//Acknowledge emergency stop
   f56_3 : BOOL ;
   A_Keyswitch0 : BOOL ;	//Keyswitch position 0
   A_Keyswitch1 : BOOL ;	//Keyswitch position 1
   A_Keyswitch2 : BOOL ;	//Keyswitch position 2
   A_Keyswitch3 : BOOL ;	//Keyswitch position 3
   A_IncInModeGroup : BOOL ;	//INC inputs in mode group area active
   f57_1 : BOOL ;
   f57_2 : BOOL ;
   A_PCshutdown : BOOL ;	//PC shutdown 840Di
   f57_4 : BOOL ;
   f57_5 : BOOL ;
   f57_6 : BOOL ;
   f57_7 : BOOL ;
   A_CollCheckOff : BOOL ;	//Collisions Check Off
   f58_1 : BOOL ;
   f58_2 : BOOL ;
   f58_3 : BOOL ;
   f58_4 : BOOL ;
   f58_5 : BOOL ;
   f58_6 : BOOL ;
   f58_7 : BOOL ;
   f59 : BYTE ;
   E_ActVal_In1 : BOOL ;	//Actual value of digi. NCK input 1
   E_ActVal_In2 : BOOL ;	//Actual value of digi. NCK input 2
   E_ActVal_In3 : BOOL ;	//Actual value of digi. NCK input 3
   E_ActVal_In4 : BOOL ;	//Actual value of digi. NCK input 4
   f60_4 : BOOL ;
   f60_5 : BOOL ;
   f60_6 : BOOL ;
   f60_7 : BOOL ;
   f61_f62 : ARRAY  [61 .. 61 ] OF BYTE ;
   E_Setpoint_Out1 : BOOL ;	//Setpoint of digi. NCK output 1
   E_Setpoint_Out2 : BOOL ;	//Setpoint of digi. NCK output 2
   E_Setpoint_Out3 : BOOL ;	//Setpoint of digi. NCK output 3
   E_Setpoint_Out4 : BOOL ;	//Setpoint of digi. NCK output 4
   E_Setpoint_Out5 : BOOL ;	//Setpoint of digi. NCK output 5
   E_Setpoint_Out6 : BOOL ;	//Setpoint of digi. NCK output 6
   E_Setpoint_Out7 : BOOL ;	//Setpoint of digi. NCK output 7
   E_Setpoint_Out8 : BOOL ;	//Setpoint of digi. NCK output 8
   f65_f67 : ARRAY  [65 .. 66 ] OF BYTE ;
   E_HW1_moved : BYTE ;	//Handwheel 1 moved
   E_HW2_moved : BYTE ;	//Handwheel 2 moved
   E_HW3_moved : BYTE ;	//Handwheel 3 moved
   E_CounterInchMetr : BYTE ;	//Modification counter inch/metric system of units
   E_MCP1AxisValid : BOOL ;	//from HT6
   E_MCP1WCS : BOOL ;	//from HT6
   f72_2 : BOOL ;
   f72_3 : BOOL ;
   f72_4 : BOOL ;
   f72_5 : BOOL ;
   f72_6 : BOOL ;
   E_MCP1AxKeyDisp : BOOL ;	//Mcp1 Axis Key Displayed
   E_MCP2AxisValid : BOOL ;	//from HT6
   E_MCP2WCS : BOOL ;	//from HT6
   f73_2 : BOOL ;
   f73_3 : BOOL ;
   f73_4 : BOOL ;
   f73_5 : BOOL ;
   f73_6 : BOOL ;
   E_MCP2AxKeyDisp : BOOL ;	//Mcp2 Axis Key Displayed
   MCP1AxisFromHMI : ARRAY  [1 .. 6 ] OF BYTE ;	//Axistable from HT6
   MCP2AxisFromHMI : ARRAY  [1 .. 6 ] OF BYTE ;	//Axistable from HT6
   res86 : WORD ;
   res88 : BYTE ;
   res89 : BYTE ;
   epsToPlc : BYTE ;
   epsFromPlc : BYTE ;
   MpiDpOk : BOOL ;	//Slaves on MPI/DP Ok
   DpOk : BOOL ;	//Slaves on DP Ok
   f92_2 : BOOL ;
   f92_3 : BOOL ;
   f92_4 : BOOL ;
   f92_5 : BOOL ;
   f92_6 : BOOL ;
   f92_7 : BOOL ;
   f93 : BYTE ;
   f94 : BYTE ;
   f95 : BYTE ;
   f96_0 : BOOL ;
   f96_1 : BOOL ;
   f96_2 : BOOL ;
   f96_3 : BOOL ;
   f96_4 : BOOL ;
   f96_5 : BOOL ;
   f96_6 : BOOL ;
   f96_7 : BOOL ;
   E_Chan_HW1_A : BOOL ;	//Channel number for handwheel1 A
   E_Chan_HW1_B : BOOL ;	//Channel number for handwheel1 B
   E_Chan_HW1_C : BOOL ;	//Channel number for handwheel1 C
   E_Chan_HW1_D : BOOL ;	//Channel number for handwheel1 D
   f97_4 : BOOL ;
   f97_5 : BOOL ;
   f97_6 : BOOL ;
   f97_7 : BOOL ;
   E_Chan_HW2_A : BOOL ;	//Channel number for handwheel2 A
   E_Chan_HW2_B : BOOL ;	//Channel number for handwheel2 B
   E_Chan_HW2_C : BOOL ;	//Channel number for handwheel2 C
   E_Chan_HW2_D : BOOL ;	//Channel number for handwheel2 D
   f98_4 : BOOL ;
   f98_5 : BOOL ;
   f98_6 : BOOL ;
   f98_7 : BOOL ;
   E_Chan_HW3_A : BOOL ;	//Channel number for handwheel3 A
   E_Chan_HW3_B : BOOL ;	//Channel number for handwheel3 B
   E_Chan_HW3_C : BOOL ;	//Channel number for handwheel3 C
   E_Chan_HW3_D : BOOL ;	//Channel number for handwheel3 D
   f99_4 : BOOL ;
   f99_5 : BOOL ;
   f99_6 : BOOL ;
   f99_7 : BOOL ;
   E_Ax_A_HW1 : BOOL ;	//Axis number for handwheel1 A
   E_Ax_B_HW1 : BOOL ;	//Axis number for handwheel1 B
   E_Ax_C_HW1 : BOOL ;	//Axis number for handwheel1 C
   E_Ax_D_HW1 : BOOL ;	//Axis number for handwheel1 D
   E_Ax_E_HW1 : BOOL ;	//Axis number for handwheel1 E
   E_CHW_sel1 : BOOL ;	//Contour handwheel selected
   E_HW_sel1 : BOOL ;	//Handwheel selected
   E_Mach_Ax1 : BOOL ;	//Machine axis
   E_Ax_A_HW2 : BOOL ;	//Axis number for handwheel2 A
   E_Ax_B_HW2 : BOOL ;	//Axis number for handwheel2 B
   E_Ax_C_HW2 : BOOL ;	//Axis number for handwheel2 C
   E_Ax_D_HW2 : BOOL ;	//Axis number for handwheel2 D
   E_Ax_E_HW2 : BOOL ;	//Axis number for handwheel2 E
   E_CHW_sel2 : BOOL ;	//Contour handwheel selected
   E_HW_sel2 : BOOL ;	//Handwheel selected
   E_Mach_Ax2 : BOOL ;	//Machine axis
   E_Ax_A_HW3 : BOOL ;	//Axis number for handwheel3 A
   E_Ax_B_HW3 : BOOL ;	//Axis number for handwheel3 B
   E_Ax_C_HW3 : BOOL ;	//Axis number for handwheel3 C
   E_Ax_D_HW3 : BOOL ;	//Axis number for handwheel3 D
   E_Ax_E_HW3 : BOOL ;	//Axis number for handwheel3 E
   E_CHW_sel3 : BOOL ;	//Contour handwheel selected
   E_HW_sel3 : BOOL ;	//Handwheel selected
   E_Mach_Ax3 : BOOL ;	//Machine axis
   E_RemDiag : BOOL ;	//Remote Diagnostic
   f103_1 : BOOL ;
   f103_2 : BOOL ;
   f103_3 : BOOL ;
   f103_4 : BOOL ;
   E_ATready : BOOL ;	//AT-box ready
   E_MMCTemp : BOOL ;	//MMC temperature limit
   E_MMCBatt : BOOL ;	//MMC 101/102 battery alarm
   E_MCP1ready : BOOL ;	//MCP1 ready;
   E_MCP2ready : BOOL ;	//MCP2 ready;
   E_BHGready : BOOL ;	//BHG ready;
   f104_3 : BOOL ;
   f104_4 : BOOL ;
   f104_5 : BOOL ;
   E_FirstOB1 : BOOL ;	//This bit is on for the first OB1 cycle
   E_NCKready : BOOL ;	//NCK CPU ready
   f105 : BYTE ;
   E_CollCheckOff : BOOL ;	//CollisionsCheck Off
   E_EMSTOP : BOOL ;	//EMERGENCY STOP active
   f106_2 : BOOL ;
   f106_3 : BOOL ;
   f106_4 : BOOL ;
   f106_5 : BOOL ;
   f106_6 : BOOL ;
   f106_7 : BOOL ;
   E_InspProbe1 : BOOL ;	//Inspection probe 1 actuated
   E_InspProbe2 : BOOL ;	//Inspection probe 2 actuated
   f107_2 : BOOL ;
   f107_3 : BOOL ;
   f107_4 : BOOL ;
   f107_5 : BOOL ;
   E_NCU_LinkActive : BOOL ;	//NCU link active
   E_SystemInchDim : BOOL ;	//System inch dimension
   f108_0 : BOOL ;
   E_MMC2Ready : BOOL ;	//MMC2-CPU ready
   E_MMCMPIready : BOOL ;	//MMC1-CPU on MPI ready
   E_MMCBTSSready : BOOL ;	//MMC1-CPU on BTSS ready
   f108_4 : BOOL ;
   E_DrivesInCylOp : BOOL ;	//Drives in cylindric operation
   E_611Dready : BOOL ;	//611D ready
   E_NCready : BOOL ;
   E_NCKalarm : BOOL ;	//NCK alarm present
   f109_1 : BOOL ;
   f109_2 : BOOL ;
   f109_3 : BOOL ;
   A_PC_OSfault : BOOL ;	//PC operating system fault, 840Di
   E_HTempAlarm : BOOL ;	//Heat sink temperature alarm NCU 573
   E_ATempAlarm : BOOL ;	//Air temperature alarm
   E_BattAlarm : BOOL ;	//NCK battery alarm
   E_SWCamMinus : ARRAY  [0 .. 31 ] OF BOOL ;	//Software cams minus [0..31]
   E_SWCamPlus : ARRAY  [0 .. 31 ] OF BOOL ;	//Software cams plus [0..31]
   f118_f121 : ARRAY  [0 .. 3 ] OF BYTE ;
   A_Disabl_Inp9 : BOOL ;	//Disable digi. NCK input 9
   A_Disabl_Inp10 : BOOL ;	//Disable digi. NCK input 10
   A_Disabl_Inp11 : BOOL ;	//Disable digi. NCK input 11
   A_Disabl_Inp12 : BOOL ;	//Disable digi. NCK input 12
   A_Disabl_Inp13 : BOOL ;	//Disable digi. NCK input 13
   A_Disabl_Inp14 : BOOL ;	//Disable digi. NCK input 14
   A_Disabl_Inp15 : BOOL ;	//Disable digi. NCK input 15
   A_Disabl_Inp16 : BOOL ;	//Disable digi. NCK input 16
   A_Set_Inp9 : BOOL ;	//Set digi. NCK input 9
   A_Set_Inp10 : BOOL ;	//Set digi. NCK input 10
   A_Set_Inp11 : BOOL ;	//Set digi. NCK input 11
   A_Set_Inp12 : BOOL ;	//Set digi. NCK input 12
   A_Set_Inp13 : BOOL ;	//Set digi. NCK input 13
   A_Set_Inp14 : BOOL ;	//Set digi. NCK input 14
   A_Set_Inp15 : BOOL ;	//Set digi. NCK input 15
   A_Set_Inp16 : BOOL ;	//Set digi. NCK input 16
   A_Disabl_Inp17 : BOOL ;	//Disable digi. NCK input 17
   A_Disabl_Inp18 : BOOL ;	//Disable digi. NCK input 18
   A_Disabl_Inp19 : BOOL ;	//Disable digi. NCK input 19
   A_Disabl_Inp20 : BOOL ;	//Disable digi. NCK input 20
   A_Disabl_Inp21 : BOOL ;	//Disable digi. NCK input 21
   A_Disabl_Inp22 : BOOL ;	//Disable digi. NCK input 22
   A_Disabl_Inp23 : BOOL ;	//Disable digi. NCK input 23
   A_Disabl_Inp24 : BOOL ;	//Disable digi. NCK input 24
   A_Set_Inp17 : BOOL ;	//Set digi. NCK input 17
   A_Set_Inp18 : BOOL ;	//Set digi. NCK input 18
   A_Set_Inp19 : BOOL ;	//Set digi. NCK input 19
   A_Set_Inp20 : BOOL ;	//Set digi. NCK input 20
   A_Set_Inp21 : BOOL ;	//Set digi. NCK input 21
   A_Set_Inp22 : BOOL ;	//Set digi. NCK input 22
   A_Set_Inp23 : BOOL ;	//Set digi. NCK input 23
   A_Set_Inp24 : BOOL ;	//Set digi. NCK input 24
   A_Disabl_Inp25 : BOOL ;	//Disable digi. NCK input 25
   A_Disabl_Inp26 : BOOL ;	//Disable digi. NCK input 26
   A_Disabl_Inp27 : BOOL ;	//Disable digi. NCK input 27
   A_Disabl_Inp28 : BOOL ;	//Disable digi. NCK input 28
   A_Disabl_Inp29 : BOOL ;	//Disable digi. NCK input 29
   A_Disabl_Inp30 : BOOL ;	//Disable digi. NCK input 30
   A_Disabl_Inp31 : BOOL ;	//Disable digi. NCK input 31
   A_Disabl_Inp32 : BOOL ;	//Disable digi. NCK input 32
   A_Set_Inp25 : BOOL ;	//Set digi. NCK input 25
   A_Set_Inp26 : BOOL ;	//Set digi. NCK input 26
   A_Set_Inp27 : BOOL ;	//Set digi. NCK input 27
   A_Set_Inp28 : BOOL ;	//Set digi. NCK input 28
   A_Set_Inp29 : BOOL ;	//Set digi. NCK input 29
   A_Set_Inp30 : BOOL ;	//Set digi. NCK input 30
   A_Set_Inp31 : BOOL ;	//Set digi. NCK input 31
   A_Set_Inp32 : BOOL ;	//Set digi. NCK input 32
   A_Disabl_Inp33 : BOOL ;	//Disable digi. NCK input 33
   A_Disabl_Inp34 : BOOL ;	//Disable digi. NCK input 34
   A_Disabl_Inp35 : BOOL ;	//Disable digi. NCK input 35
   A_Disabl_Inp36 : BOOL ;	//Disable digi. NCK input 36
   A_Disabl_Inp37 : BOOL ;	//Disable digi. NCK input 37
   A_Disabl_Inp38 : BOOL ;	//Disable digi. NCK input 38
   A_Disabl_Inp39 : BOOL ;	//Disable digi. NCK input 39
   A_Disabl_Inp40 : BOOL ;	//Disable digi. NCK input 40
   A_Set_Inp33 : BOOL ;	//Set digi. NCK input 33
   A_Set_Inp34 : BOOL ;	//Set digi. NCK input 34
   A_Set_Inp35 : BOOL ;	//Set digi. NCK input 35
   A_Set_Inp36 : BOOL ;	//Set digi. NCK input 36
   A_Set_Inp37 : BOOL ;	//Set digi. NCK input 37
   A_Set_Inp38 : BOOL ;	//Set digi. NCK input 38
   A_Set_Inp39 : BOOL ;	//Set digi. NCK input 39
   A_Set_Inp40 : BOOL ;	//Set digi. NCK input 40
   A_Disabl_Out9 : BOOL ;	//Disable digi. NCK output 9
   A_Disabl_Out10 : BOOL ;	//Disable digi. NCK output 10
   A_Disabl_Out11 : BOOL ;	//Disable digi. NCK output 11
   A_Disabl_Out12 : BOOL ;	//Disable digi. NCK output 12
   A_Disabl_Out13 : BOOL ;	//Disable digi. NCK output 13
   A_Disabl_Out14 : BOOL ;	//Disable digi. NCK output 14
   A_Disabl_Out15 : BOOL ;	//Disable digi. NCK output 15
   A_Disabl_Out16 : BOOL ;	//Disable digi. NCK output 16
   A_OvMask_Out9 : BOOL ;	//Overwrite mask of digi. output 9
   A_OvMask_Out10 : BOOL ;	//Overwrite mask of digi. output 10
   A_OvMask_Out11 : BOOL ;	//Overwrite mask of digi. output 11
   A_OvMask_Out12 : BOOL ;	//Overwrite mask of digi. output 12
   A_OvMask_Out13 : BOOL ;	//Overwrite mask of digi. output 13
   A_OvMask_Out14 : BOOL ;	//Overwrite mask of digi. output 14
   A_OvMask_Out15 : BOOL ;	//Overwrite mask of digi. output 15
   A_OvMask_Out16 : BOOL ;	//Overwrite mask of digi. output 16
   A_Setval_Out9 : BOOL ;	//Set value digi. NCK output 9
   A_Setval_Out10 : BOOL ;	//Set value digi. NCK output 10
   A_Setval_Out11 : BOOL ;	//Set value digi. NCK output 11
   A_Setval_Out12 : BOOL ;	//Set value digi. NCK output 12
   A_Setval_Out13 : BOOL ;	//Set value digi. NCK output 13
   A_Setval_Out14 : BOOL ;	//Set value digi. NCK output 14
   A_Setval_Out15 : BOOL ;	//Set value digi. NCK output 15
   A_Setval_Out16 : BOOL ;	//Set value digi. NCK output 16
   A_InMask_Out9 : BOOL ;	//Input mask of digi. output 9
   A_InMask_Out10 : BOOL ;	//Input mask of digi. output 10
   A_InMask_Out11 : BOOL ;	//Input mask of digi. output 11
   A_InMask_Out12 : BOOL ;	//Input mask of digi. output 12
   A_InMask_Out13 : BOOL ;	//Input mask of digi. output 13
   A_InMask_Out14 : BOOL ;	//Input mask of digi. output 14
   A_InMask_Out15 : BOOL ;	//Input mask of digi. output 15
   A_InMask_Out16 : BOOL ;	//Input mask of digi. output 16
   A_Disabl_Out17 : BOOL ;	//Disable digi. NCK output 17
   A_Disabl_Out18 : BOOL ;	//Disable digi. NCK output 18
   A_Disabl_Out19 : BOOL ;	//Disable digi. NCK output 19
   A_Disabl_Out20 : BOOL ;	//Disable digi. NCK output 20
   A_Disabl_Out21 : BOOL ;	//Disable digi. NCK output 21
   A_Disabl_Out22 : BOOL ;	//Disable digi. NCK output 22
   A_Disabl_Out23 : BOOL ;	//Disable digi. NCK output 23
   A_Disabl_Out24 : BOOL ;	//Disable digi. NCK output 24
   A_OvMask_Out17 : BOOL ;	//Overwrite mask of digi. output 17
   A_OvMask_Out18 : BOOL ;	//Overwrite mask of digi. output 18
   A_OvMask_Out19 : BOOL ;	//Overwrite mask of digi. output 19
   A_OvMask_Out20 : BOOL ;	//Overwrite mask of digi. output 20
   A_OvMask_Out21 : BOOL ;	//Overwrite mask of digi. output 21
   A_OvMask_Out22 : BOOL ;	//Overwrite mask of digi. output 22
   A_OvMask_Out23 : BOOL ;	//Overwrite mask of digi. output 23
   A_OvMask_Out24 : BOOL ;	//Overwrite mask of digi. output 24
   A_Setval_Out17 : BOOL ;	//Set value digi. NCK output 17
   A_Setval_Out18 : BOOL ;	//Set value digi. NCK output 18
   A_Setval_Out19 : BOOL ;	//Set value digi. NCK output 19
   A_Setval_Out20 : BOOL ;	//Set value digi. NCK output 20
   A_Setval_Out21 : BOOL ;	//Set value digi. NCK output 21
   A_Setval_Out22 : BOOL ;	//Set value digi. NCK output 22
   A_Setval_Out23 : BOOL ;	//Set value digi. NCK output 23
   A_Setval_Out24 : BOOL ;	//Set value digi. NCK output 24
   A_InMask_Out17 : BOOL ;	//Input mask of digi. output 17
   A_InMask_Out18 : BOOL ;	//Input mask of digi. output 18
   A_InMask_Out19 : BOOL ;	//Input mask of digi. output 19
   A_InMask_Out20 : BOOL ;	//Input mask of digi. output 20
   A_InMask_Out21 : BOOL ;	//Input mask of digi. output 21
   A_InMask_Out22 : BOOL ;	//Input mask of digi. output 22
   A_InMask_Out23 : BOOL ;	//Input mask of digi. output 23
   A_InMask_Out24 : BOOL ;	//Input mask of digi. output 24
   A_Disabl_Out25 : BOOL ;	//Disable digi. NCK output 25
   A_Disabl_Out26 : BOOL ;	//Disable digi. NCK output 26
   A_Disabl_Out27 : BOOL ;	//Disable digi. NCK output 27
   A_Disabl_Out28 : BOOL ;	//Disable digi. NCK output 28
   A_Disabl_Out29 : BOOL ;	//Disable digi. NCK output 29
   A_Disabl_Out30 : BOOL ;	//Disable digi. NCK output 30
   A_Disabl_Out31 : BOOL ;	//Disable digi. NCK output 31
   A_Disabl_Out32 : BOOL ;	//Disable digi. NCK output 32
   A_OvMask_Out25 : BOOL ;	//Overwrite mask of digi. output 25
   A_OvMask_Out26 : BOOL ;	//Overwrite mask of digi. output 26
   A_OvMask_Out27 : BOOL ;	//Overwrite mask of digi. output 27
   A_OvMask_Out28 : BOOL ;	//Overwrite mask of digi. output 28
   A_OvMask_Out29 : BOOL ;	//Overwrite mask of digi. output 29
   A_OvMask_Out30 : BOOL ;	//Overwrite mask of digi. output 30
   A_OvMask_Out31 : BOOL ;	//Overwrite mask of digi. output 31
   A_OvMask_Out32 : BOOL ;	//Overwrite mask of digi. output 32
   A_Setval_Out25 : BOOL ;	//Set value digi. NCK output 25
   A_Setval_Out26 : BOOL ;	//Set value digi. NCK output 26
   A_Setval_Out27 : BOOL ;	//Set value digi. NCK output 27
   A_Setval_Out28 : BOOL ;	//Set value digi. NCK output 28
   A_Setval_Out29 : BOOL ;	//Set value digi. NCK output 29
   A_Setval_Out30 : BOOL ;	//Set value digi. NCK output 30
   A_Setval_Out31 : BOOL ;	//Set value digi. NCK output 31
   A_Setval_Out32 : BOOL ;	//Set value digi. NCK output 32
   A_InMask_Out25 : BOOL ;	//Input mask of digi. output 25
   A_InMask_Out26 : BOOL ;	//Input mask of digi. output 26
   A_InMask_Out27 : BOOL ;	//Input mask of digi. output 27
   A_InMask_Out28 : BOOL ;	//Input mask of digi. output 28
   A_InMask_Out29 : BOOL ;	//Input mask of digi. output 29
   A_InMask_Out30 : BOOL ;	//Input mask of digi. output 30
   A_InMask_Out31 : BOOL ;	//Input mask of digi. output 31
   A_InMask_Out32 : BOOL ;	//Input mask of digi. output 32
   A_Disabl_Out33 : BOOL ;	//Disable digi. NCK output 33
   A_Disabl_Out34 : BOOL ;	//Disable digi. NCK output 34
   A_Disabl_Out35 : BOOL ;	//Disable digi. NCK output 35
   A_Disabl_Out36 : BOOL ;	//Disable digi. NCK output 36
   A_Disabl_Out37 : BOOL ;	//Disable digi. NCK output 37
   A_Disabl_Out38 : BOOL ;	//Disable digi. NCK output 38
   A_Disabl_Out39 : BOOL ;	//Disable digi. NCK output 39
   A_Disabl_Out40 : BOOL ;	//Disable digi. NCK output 40
   A_OvMask_Out33 : BOOL ;	//Overwrite mask of digi. output 33
   A_OvMask_Out34 : BOOL ;	//Overwrite mask of digi. output 34
   A_OvMask_Out35 : BOOL ;	//Overwrite mask of digi. output 35
   A_OvMask_Out36 : BOOL ;	//Overwrite mask of digi. output 36
   A_OvMask_Out37 : BOOL ;	//Overwrite mask of digi. output 37
   A_OvMask_Out38 : BOOL ;	//Overwrite mask of digi. output 38
   A_OvMask_Out39 : BOOL ;	//Overwrite mask of digi. output 39
   A_OvMask_Out40 : BOOL ;	//Overwrite mask of digi. output 40
   A_Setval_out33 : BOOL ;	//Set value digi. NCK output 33
   A_Setval_out34 : BOOL ;	//Set value digi. NCK output 34
   A_Setval_out35 : BOOL ;	//Set value digi. NCK output 35
   A_Setval_out36 : BOOL ;	//Set value digi. NCK output 36
   A_Setval_out37 : BOOL ;	//Set value digi. NCK output 37
   A_Setval_out38 : BOOL ;	//Set value digi. NCK output 38
   A_Setval_out39 : BOOL ;	//Set value digi. NCK output 39
   A_Setval_out40 : BOOL ;	//Set value digi. NCK output 40
   A_InMask_Out33 : BOOL ;	//Input mask of digi. output 33
   A_InMask_Out34 : BOOL ;	//Input mask of digi. output 34
   A_InMask_Out35 : BOOL ;	//Input mask of digi. output 35
   A_InMask_Out36 : BOOL ;	//Input mask of digi. output 36
   A_InMask_Out37 : BOOL ;	//Input mask of digi. output 37
   A_InMask_Out38 : BOOL ;	//Input mask of digi. output 38
   A_InMask_Out39 : BOOL ;	//Input mask of digi. output 39
   A_InMask_Out40 : BOOL ;	//Input mask of digi. output 40
   A_Disabl_anaIn1 : BOOL ;	//Disable analog NCK input 1
   A_Disabl_anaIn2 : BOOL ;	//Disable analog NCK input 2
   A_Disabl_anaIn3 : BOOL ;	//Disable analog NCK input 3
   A_Disabl_anaIn4 : BOOL ;	//Disable analog NCK input 4
   A_Disabl_anaIn5 : BOOL ;	//Disable analog NCK input 5
   A_Disabl_anaIn6 : BOOL ;	//Disable analog NCK input 6
   A_Disabl_anaIn7 : BOOL ;	//Disable analog NCK input 7
   A_Disabl_anaIn8 : BOOL ;	//Disable analog NCK input 8
   A_InMask_anaIn1 : BOOL ;	//Input mask of analog NCK input 1
   A_InMask_anaIn2 : BOOL ;	//Input mask of analog NCK input 2
   A_InMask_anaIn3 : BOOL ;	//Input mask of analog NCK input 3
   A_InMask_anaIn4 : BOOL ;	//Input mask of analog NCK input 4
   A_InMask_anaIn5 : BOOL ;	//Input mask of analog NCK input 5
   A_InMask_anaIn6 : BOOL ;	//Input mask of analog NCK input 6
   A_InMask_anaIn7 : BOOL ;	//Input mask of analog NCK input 7
   A_InMask_anaIn8 : BOOL ;	//Input mask of analog NCK input 8
   A_Setval_anaIn1 : WORD ;	//Set value of analog NCK input 1
   A_Setval_anaIn2 : WORD ;	//Set value of analog NCK input 2
   A_Setval_anaIn3 : WORD ;	//Set value of analog NCK input 3
   A_Setval_anaIn4 : WORD ;	//Set value of analog NCK input 4
   A_Setval_anaIn5 : WORD ;	//Set value of analog NCK input 5
   A_Setval_anaIn6 : WORD ;	//Set value of analog NCK input 6
   A_Setval_anaIn7 : WORD ;	//Set value of analog NCK input 7
   A_Setval_anaIn8 : WORD ;	//Set value of analog NCK input 8
   f164_f165 : INT ;
   A_OvMask_anaOut1 : BOOL ;	//Overwrite mask of analog output 1
   A_OvMask_anaOut2 : BOOL ;	//Overwrite mask of analog output 2
   A_OvMask_anaOut3 : BOOL ;	//Overwrite mask of analog output 3
   A_OvMask_anaOut4 : BOOL ;	//Overwrite mask of analog output 4
   A_OvMask_anaOut5 : BOOL ;	//Overwrite mask of analog output 5
   A_OvMask_anaOut6 : BOOL ;	//Overwrite mask of analog output 6
   A_OvMask_anaOut7 : BOOL ;	//Overwrite mask of analog output 7
   A_OvMask_anaOut8 : BOOL ;	//Overwrite mask of analog output 8
   A_InMask_anaOut1 : BOOL ;	//Input mask of analog NCK output 1
   A_InMask_anaOut2 : BOOL ;	//Input mask of analog NCK output 2
   A_InMask_anaOut3 : BOOL ;	//Input mask of analog NCK output 3
   A_InMask_anaOut4 : BOOL ;	//Input mask of analog NCK output 4
   A_InMask_anaOut5 : BOOL ;	//Input mask of analog NCK output 5
   A_InMask_anaOut6 : BOOL ;	//Input mask of analog NCK output 6
   A_InMask_anaOut7 : BOOL ;	//Input mask of analog NCK output 7
   A_InMask_anaOut8 : BOOL ;	//Input mask of analog NCK output 8
   A_Disabl_anaOut1 : BOOL ;	//Disable analog NCK output 1
   A_Disabl_anaOut2 : BOOL ;	//Disable analog NCK output 2
   A_Disabl_anaOut3 : BOOL ;	//Disable analog NCK output 3
   A_Disabl_anaOut4 : BOOL ;	//Disable analog NCK output 4
   A_Disabl_anaOut5 : BOOL ;	//Disable analog NCK output 5
   A_Disabl_anaOut6 : BOOL ;	//Disable analog NCK output 6
   A_Disabl_anaOut7 : BOOL ;	//Disable analog NCK output 7
   A_Disabl_anaOut8 : BOOL ;	//Disable analog NCK output 8
   f169 : BYTE ;
   A_Setval_anaOut1 : WORD ;	//Set value of analog NCK output 1
   A_Setval_anaOut2 : WORD ;	//Set value of analog NCK output 2
   A_Setval_anaOut3 : WORD ;	//Set value of analog NCK output 3
   A_Setval_anaOut4 : WORD ;	//Set value of analog NCK output 4
   A_Setval_anaOut5 : WORD ;	//Set value of analog NCK output 5
   A_Setval_anaOut6 : WORD ;	//Set value of analog NCK output 6
   A_Setval_anaOut7 : WORD ;	//Set value of analog NCK output 7
   A_Setval_anaOut8 : WORD ;	//Set value of analog NCK output 8
   E_ActVal_In9 : BOOL ;	//Actual value of digi. NCK input 9
   E_ActVal_In10 : BOOL ;	//Actual value of digi. NCK input 10
   E_ActVal_In11 : BOOL ;	//Actual value of digi. NCK input 11
   E_ActVal_In12 : BOOL ;	//Actual value of digi. NCK input 12
   E_ActVal_In13 : BOOL ;	//Actual value of digi. NCK input 13
   E_ActVal_In14 : BOOL ;	//Actual value of digi. NCK input 14
   E_ActVal_In15 : BOOL ;	//Actual value of digi. NCK input 15
   E_ActVal_In16 : BOOL ;	//Actual value of digi. NCK input 16
   E_ActVal_In17 : BOOL ;	//Actual value of digi. NCK input 17
   E_ActVal_In18 : BOOL ;	//Actual value of digi. NCK input 18
   E_ActVal_In19 : BOOL ;	//Actual value of digi. NCK input 19
   E_ActVal_In20 : BOOL ;	//Actual value of digi. NCK input 20
   E_ActVal_In21 : BOOL ;	//Actual value of digi. NCK input 21
   E_ActVal_In22 : BOOL ;	//Actual value of digi. NCK input 22
   E_ActVal_In23 : BOOL ;	//Actual value of digi. NCK input 23
   E_ActVal_In24 : BOOL ;	//Actual value of digi. NCK input 24
   E_ActVal_In25 : BOOL ;	//Actual value of digi. NCK input 25
   E_ActVal_In26 : BOOL ;	//Actual value of digi. NCK input 26
   E_ActVal_In27 : BOOL ;	//Actual value of digi. NCK input 27
   E_ActVal_In28 : BOOL ;	//Actual value of digi. NCK input 28
   E_ActVal_In29 : BOOL ;	//Actual value of digi. NCK input 29
   E_ActVal_In30 : BOOL ;	//Actual value of digi. NCK input 30
   E_ActVal_In31 : BOOL ;	//Actual value of digi. NCK input 31
   E_ActVal_In32 : BOOL ;	//Actual value of digi. NCK input 32
   E_ActVal_In33 : BOOL ;	//Actual value of digi. NCK input 33
   E_ActVal_In34 : BOOL ;	//Actual value of digi. NCK input 34
   E_ActVal_In35 : BOOL ;	//Actual value of digi. NCK input 35
   E_ActVal_In36 : BOOL ;	//Actual value of digi. NCK input 36
   E_ActVal_In37 : BOOL ;	//Actual value of digi. NCK input 37
   E_ActVal_In38 : BOOL ;	//Actual value of digi. NCK input 38
   E_ActVal_In39 : BOOL ;	//Actual value of digi. NCK input 39
   E_ActVal_In40 : BOOL ;	//Actual value of digi. NCK input 40
   E_Setpoint_Out9 : BOOL ;	//Setpoint of digi. NCK output 9
   E_Setpoint_Out10 : BOOL ;	//Setpoint of digi. NCK output 10
   E_Setpoint_Out11 : BOOL ;	//Setpoint of digi. NCK output 11
   E_Setpoint_Out12 : BOOL ;	//Setpoint of digi. NCK output 12
   E_Setpoint_Out13 : BOOL ;	//Setpoint of digi. NCK output 13
   E_Setpoint_Out14 : BOOL ;	//Setpoint of digi. NCK output 14
   E_Setpoint_Out15 : BOOL ;	//Setpoint of digi. NCK output 15
   E_Setpoint_Out16 : BOOL ;	//Setpoint of digi. NCK output 16
   E_Setpoint_Out17 : BOOL ;	//Setpoint of digi. NCK output 17
   E_Setpoint_Out18 : BOOL ;	//Setpoint of digi. NCK output 18
   E_Setpoint_Out19 : BOOL ;	//Setpoint of digi. NCK output 19
   E_Setpoint_Out20 : BOOL ;	//Setpoint of digi. NCK output 20
   E_Setpoint_Out21 : BOOL ;	//Setpoint of digi. NCK output 21
   E_Setpoint_Out22 : BOOL ;	//Setpoint of digi. NCK output 22
   E_Setpoint_Out23 : BOOL ;	//Setpoint of digi. NCK output 23
   E_Setpoint_Out24 : BOOL ;	//Setpoint of digi. NCK output 24
   E_Setpoint_Out25 : BOOL ;	//Setpoint of digi. NCK output 25
   E_Setpoint_Out26 : BOOL ;	//Setpoint of digi. NCK output 26
   E_Setpoint_Out27 : BOOL ;	//Setpoint of digi. NCK output 27
   E_Setpoint_Out28 : BOOL ;	//Setpoint of digi. NCK output 28
   E_Setpoint_Out29 : BOOL ;	//Setpoint of digi. NCK output 29
   E_Setpoint_Out30 : BOOL ;	//Setpoint of digi. NCK output 30
   E_Setpoint_Out31 : BOOL ;	//Setpoint of digi. NCK output 31
   E_Setpoint_Out32 : BOOL ;	//Setpoint of digi. NCK output 32
   E_Setpoint_Out33 : BOOL ;	//Setpoint of digi. NCK output 33
   E_Setpoint_Out34 : BOOL ;	//Setpoint of digi. NCK output 34
   E_Setpoint_Out35 : BOOL ;	//Setpoint of digi. NCK output 35
   E_Setpoint_Out36 : BOOL ;	//Setpoint of digi. NCK output 36
   E_Setpoint_Out37 : BOOL ;	//Setpoint of digi. NCK output 37
   E_Setpoint_Out38 : BOOL ;	//Setpoint of digi. NCK output 38
   E_Setpoint_Out39 : BOOL ;	//Setpoint of digi. NCK output 39
   E_Setpoint_Out40 : BOOL ;	//Setpoint of digi. NCK output 40
   E_ActVal_anaIn1 : WORD ;	//Actual value of analog NCK input 1
   E_ActVal_anaIn2 : WORD ;	//Actual value of analog NCK input 2
   E_ActVal_anaIn3 : WORD ;	//Actual value of analog NCK input 3
   E_ActVal_anaIn4 : WORD ;	//Actual value of analog NCK input 4
   E_ActVal_anaIn5 : WORD ;	//Actual value of analog NCK input 5
   E_ActVal_anaIn6 : WORD ;	//Actual value of analog NCK input 6
   E_ActVal_anaIn7 : WORD ;	//Actual value of analog NCK input 7
   E_ActVal_anaIn8 : WORD ;	//Actual value of analog NCK input 8
   E_SetVal_anaOut1 : WORD ;	//Set value of analog NCK output 1
   E_SetVal_anaOut2 : WORD ;	//Set value of analog NCK output 2
   E_SetVal_anaOut3 : WORD ;	//Set value of analog NCK output 3
   E_SetVal_anaOut4 : WORD ;	//Set value of analog NCK output 4
   E_SetVal_anaOut5 : WORD ;	//Set value of analog NCK output 5
   E_SetVal_anaOut6 : WORD ;	//Set value of analog NCK output 6
   E_SetVal_anaOut7 : WORD ;	//Set value of analog NCK output 7
   E_SetVal_anaOut8 : WORD ;	//Set value of analog NCK output 8
   E_CollCheck : ARRAY  [0 .. 7 ] OF BYTE ;	//CollisionsCheck
   A_CollCheck : ARRAY  [0 .. 7 ] OF BYTE ;	//CollisionsCheck
  END_STRUCT ;	
END_TYPE

